C07281=1059.069,212.928,410.818,172.562,33.057,156.142
C07282=1059.063,212.678,410.844,172.560,33.053,156.141
C07283=1059.056,212.430,410.870,172.558,33.049,156.141
C07284=1059.050,212.181,410.896,172.556,33.045,156.140
C07285=1059.045,211.932,410.922,172.554,33.041,156.139
C07286=1059.038,211.684,410.948,172.552,33.037,156.138
C07287=1059.032,211.436,410.973,172.550,33.033,156.138
C07288=1059.026,211.187,411.000,172.548,33.029,156.137
C07289=1059.020,210.939,411.025,172.546,33.026,156.136
C07290=1059.013,210.690,411.051,172.544,33.022,156.135
C07291=1059.007,210.441,411.077,172.542,33.018,156.135
C07292=1059.001,210.192,411.103,172.540,33.014,156.134
C07293=1058.995,209.944,411.129,172.538,33.010,156.133
C07294=1058.988,209.696,411.154,172.536,33.006,156.132
C07295=1058.983,209.447,411.180,172.534,33.002,156.132
C07296=1058.976,209.199,411.206,172.532,32.998,156.131
C07297=1058.970,208.950,411.231,172.530,32.994,156.130
C07298=1058.965,208.717,411.256,172.529,32.990,156.130
C07299=1058.959,208.484,411.280,172.527,32.986,156.129
C07300=1058.954,208.252,411.304,172.525,32.983,156.128
C07301=1058.947,208.020,411.328,172.523,32.979,156.127
C07302=1058.941,207.788,411.352,172.521,32.975,156.127
C07303=1058.936,207.555,411.376,172.520,32.972,156.126
C07304=1058.930,207.323,411.400,172.518,32.968,156.125
C07305=1058.924,207.090,411.424,172.516,32.964,156.125
C07306=1058.899,206.041,411.528,172.330,32.878,156.114
C07307=1058.893,205.792,411.553,172.327,32.874,156.114
C07308=1058.888,205.543,411.577,172.325,32.871,156.113
C07309=1058.881,205.295,411.602,172.323,32.868,156.113
C07310=1058.875,205.045,411.627,172.320,32.865,156.112
C07311=1058.870,204.797,411.652,172.318,32.862,156.112
C07312=1058.864,204.548,411.677,172.316,32.859,156.111
C07313=1058.858,204.300,411.702,172.313,32.856,156.110
C07314=1058.852,204.051,411.726,172.311,32.853,156.110
C07315=1058.846,203.802,411.750,172.309,32.850,156.109
C07316=1058.840,203.554,411.775,172.306,32.846,156.109
C07317=1058.834,203.304,411.800,172.304,32.843,156.108
C07318=1058.829,203.056,411.824,172.302,32.841,156.108
C07319=1058.823,202.807,411.849,172.299,32.838,156.107
C07320=1058.817,202.559,411.874,172.297,32.834,156.107
C07321=1058.811,202.310,411.898,172.295,32.831,156.106
C07322=1058.805,202.062,411.923,172.292,32.828,156.106
C07323=1058.799,201.812,411.947,172.290,32.825,156.105
C07324=1058.793,201.563,411.972,172.288,32.822,156.105
C07325=1058.787,201.315,411.996,172.285,32.819,156.104
C07326=1058.781,201.066,412.020,172.283,32.816,156.104
C07327=1058.775,200.818,412.045,172.281,32.813,156.103
C07328=1058.769,200.569,412.069,172.278,32.810,156.103
C07329=1058.763,200.320,412.093,172.276,32.807,156.102
C07330=1058.757,200.071,412.117,172.274,32.804,156.102
C07331=1058.751,199.822,412.142,172.271,32.801,156.101
C07332=1058.745,199.573,412.166,172.269,32.798,156.100
C07333=1058.739,199.325,412.191,172.267,32.796,156.100
C07334=1058.733,199.077,412.215,172.265,32.792,156.099
C07335=1058.727,198.827,412.239,172.262,32.789,156.099
C07336=1058.721,198.579,412.263,172.260,32.787,156.098
C07337=1058.715,198.330,412.288,172.258,32.783,156.098
C07338=1058.709,198.081,412.311,172.255,32.780,156.097
C07339=1058.703,197.832,412.336,172.253,32.778,156.097
C07340=1058.697,197.584,412.360,172.251,32.775,156.096
C07341=1058.691,197.335,412.384,172.248,32.771,156.096
C07342=1058.685,197.086,412.408,172.247,32.769,156.095
C07343=1058.679,196.837,412.432,172.245,32.766,156.095
C07344=1058.674,196.588,412.457,172.243,32.762,156.094
C07345=1058.668,196.339,412.481,172.240,32.760,156.094
C07346=1058.662,196.091,412.505,172.238,32.757,156.093
C07347=1058.656,195.843,412.529,172.236,32.754,156.093
C07348=1058.650,195.593,412.553,172.234,32.751,156.092
C07349=1058.644,195.345,412.577,172.231,32.748,156.092
C07350=1058.638,195.096,412.602,172.229,32.745,156.091
C07351=1058.632,194.847,412.625,172.227,32.742,156.091
C07352=1058.626,194.598,412.650,172.224,32.739,156.090
C07353=1058.620,194.350,412.674,172.222,32.736,156.090
C07354=1058.615,194.101,412.698,172.220,32.733,156.089
C07355=1058.608,193.852,412.722,172.218,32.730,156.089
C07356=1058.603,193.604,412.746,172.215,32.727,156.088
C07357=1058.597,193.355,412.770,172.213,32.724,156.088
C07358=1058.592,193.106,412.794,172.211,32.722,156.087
C07359=1058.586,192.857,412.817,172.209,32.718,156.087
C07360=1058.579,192.608,412.841,172.207,32.715,156.086
C07361=1058.574,192.360,412.866,172.204,32.713,156.086
C07362=1058.568,192.111,412.889,172.202,32.709,156.085
C07363=1058.562,191.862,412.914,172.200,32.707,156.085
C07364=1058.556,191.613,412.937,172.198,32.704,156.084
C07365=1058.551,191.365,412.961,172.195,32.700,156.084
C07366=1058.544,191.116,412.985,172.193,32.698,156.083
C07367=1058.538,190.832,413.012,172.191,32.695,156.083
C07368=1058.531,190.548,413.040,172.188,32.691,156.082
C07369=1058.525,190.265,413.066,172.186,32.688,156.081
C07370=1058.518,189.981,413.094,172.184,32.684,156.081
C07371=1058.511,189.732,413.118,172.182,32.681,156.080
C07372=1058.507,189.483,413.142,172.180,32.679,156.080
C07373=1058.500,189.235,413.165,172.177,32.675,156.079
C07374=1058.494,188.986,413.189,172.175,32.672,156.079
C07375=1058.489,188.736,413.213,172.173,32.670,156.078
C07376=1058.483,188.488,413.237,172.171,32.667,156.078
C07377=1058.478,188.240,413.261,172.169,32.664,156.077
C07378=1058.471,187.990,413.284,172.166,32.661,156.077
C07379=1058.466,187.741,413.308,172.164,32.658,156.076
C07380=1058.460,187.493,413.332,172.162,32.655,156.076
C07381=1058.454,187.244,413.355,172.160,32.652,156.075
C07382=1058.449,186.996,413.379,172.158,32.649,156.075
C07383=1058.442,186.746,413.403,172.156,32.646,156.074
C07384=1058.437,186.497,413.427,172.153,32.644,156.074
C07385=1058.431,186.249,413.450,172.151,32.640,156.073
C07386=1058.425,186.000,413.473,172.149,32.638,156.073
C07387=1058.420,185.752,413.498,172.147,32.635,156.072
C07388=1058.414,185.502,413.521,172.145,32.631,156.072
C07389=1058.408,185.253,413.545,172.143,32.629,156.071
C07390=1058.403,185.005,413.568,172.140,32.626,156.071
C07391=1058.397,184.756,413.592,172.138,32.623,156.070
C07392=1058.392,184.507,413.615,172.136,32.620,156.070
C07393=1058.385,184.258,413.639,172.134,32.617,156.069
C07394=1058.379,184.009,413.662,172.133,32.614,156.069
C07395=1058.373,183.761,413.686,172.131,32.612,156.068
C07396=1058.367,183.511,413.709,172.128,32.609,156.068
C07397=1058.361,183.262,413.732,172.126,32.606,156.068
C07398=1058.355,183.014,413.756,172.124,32.603,156.067
C07399=1058.349,182.765,413.779,172.122,32.601,156.067
C07400=1058.343,182.516,413.802,172.120,32.598,156.066
C07401=1058.336,182.268,413.825,172.118,32.595,156.066
C07402=1058.331,182.019,413.848,172.115,32.592,156.065
C07403=1058.325,181.770,413.871,172.113,32.590,156.065
C07404=1058.318,181.521,413.895,172.111,32.587,156.064
C07405=1058.313,181.272,413.918,172.109,32.584,156.064
C07406=1058.307,181.023,413.941,172.107,32.581,156.063
C07407=1058.301,180.775,413.965,172.105,32.579,156.063
C07408=1058.294,180.525,413.988,172.102,32.576,156.063
C07409=1058.289,180.276,414.011,172.100,32.573,156.062
C07410=1058.283,180.027,414.034,172.098,32.570,156.062
C07411=1058.276,179.779,414.057,172.096,32.568,156.061
C07412=1058.270,179.531,414.080,172.094,32.565,156.061
C07413=1058.264,179.281,414.103,172.092,32.562,156.060
C07414=1058.258,179.032,414.126,172.090,32.559,156.060
C07415=1058.252,178.784,414.150,172.088,32.557,156.059
C07416=1058.247,178.535,414.173,172.086,32.554,156.059
C07417=1058.241,178.286,414.196,172.084,32.551,156.058
C07418=1058.235,178.037,414.219,172.082,32.548,156.058
C07419=1058.228,177.788,414.241,172.080,32.546,156.057
C07420=1058.222,177.539,414.264,172.078,32.543,156.057
C07421=1058.216,177.291,414.288,172.076,32.540,156.056
C07422=1058.211,177.042,414.311,172.073,32.537,156.056
C07423=1058.205,176.793,414.334,172.071,32.535,156.056
C07424=1058.199,176.544,414.357,172.069,32.532,156.055
C07425=1058.193,176.295,414.380,172.067,32.529,156.055
C07426=1058.186,176.046,414.403,172.065,32.527,156.054
C07427=1058.181,175.797,414.426,172.063,32.524,156.054
C07428=1058.175,175.548,414.448,172.061,32.521,156.053
C07429=1058.169,175.299,414.471,172.059,32.518,156.053
C07430=1058.163,175.050,414.494,172.057,32.516,156.052
C07431=1058.156,174.766,414.521,172.054,32.512,156.052
C07432=1058.149,174.482,414.546,172.052,32.509,156.051
C07433=1058.143,174.198,414.573,172.050,32.506,156.051
C07434=1058.137,173.914,414.599,172.048,32.503,156.050
C07435=1058.131,173.665,414.622,172.046,32.500,156.050
C07436=1058.125,173.416,414.645,172.044,32.498,156.049
C07437=1058.118,173.167,414.667,172.042,32.495,156.049
C07438=1058.112,172.918,414.690,172.040,32.492,156.048
C07439=1058.107,172.669,414.713,172.038,32.489,156.048
C07440=1058.101,172.420,414.736,172.036,32.487,156.047
C07441=1058.095,172.171,414.759,172.034,32.483,156.047
C07442=1058.089,171.923,414.781,172.031,32.481,156.047
C07443=1058.083,171.674,414.804,172.029,32.478,156.046
C07444=1058.077,171.425,414.827,172.027,32.476,156.046
C07445=1058.071,171.176,414.850,172.025,32.472,156.045
C07446=1058.066,170.927,414.873,172.023,32.470,156.045
C07447=1058.059,170.679,414.896,172.021,32.467,156.044
C07448=1058.054,170.429,414.918,172.019,32.465,156.044
C07449=1058.048,170.180,414.941,172.017,32.461,156.043
C07450=1058.042,169.931,414.964,172.015,32.459,156.043
C07451=1058.037,169.682,414.987,172.014,32.456,156.042
C07452=1058.031,169.435,415.009,172.012,32.454,156.042
C07453=1058.025,169.186,415.032,172.010,32.451,156.041
C07454=1058.020,168.936,415.054,172.008,32.448,156.041
C07455=1058.014,168.687,415.077,172.006,32.445,156.041
C07456=1058.007,168.439,415.099,172.004,32.443,156.040
C07457=1058.002,168.190,415.122,172.002,32.440,156.040
C07458=1057.996,167.941,415.145,172.000,32.437,156.039
C07459=1057.991,167.691,415.167,171.998,32.434,156.039
C07460=1057.985,167.442,415.190,171.996,32.432,156.038
C07461=1057.978,167.194,415.213,171.994,32.429,156.038
C07462=1057.973,166.945,415.235,171.992,32.426,156.037
C07463=1057.967,166.695,415.258,171.989,32.423,156.037
C07464=1057.962,166.447,415.280,171.987,32.421,156.036
C07465=1057.956,166.199,415.303,171.985,32.418,156.036
C07466=1057.950,165.949,415.325,171.983,32.415,156.036
C07467=1057.944,165.700,415.348,171.982,32.412,156.035
C07468=1057.938,165.452,415.370,171.980,32.410,156.035
C07469=1057.933,165.202,415.392,171.978,32.407,156.034
C07470=1057.927,164.953,415.415,171.976,32.404,156.034
C07471=1057.921,164.704,415.438,171.974,32.401,156.033
C07472=1057.916,164.456,415.460,171.972,32.399,156.033
C07473=1057.910,164.207,415.483,171.970,32.396,156.032
C07474=1057.904,163.958,415.505,171.968,32.393,156.032
C07475=1057.899,163.709,415.528,171.966,32.391,156.031
C07476=1057.892,163.460,415.550,171.964,32.388,156.031
C07477=1057.887,163.212,415.573,171.962,32.385,156.030
C07478=1057.882,162.962,415.595,171.960,32.382,156.030
C07479=1057.875,162.714,415.617,171.958,32.380,156.030
C07480=1057.870,162.464,415.639,171.956,32.376,156.029
C07481=1057.864,162.215,415.662,171.954,32.374,156.029
C07482=1057.859,161.966,415.684,171.952,32.371,156.028
C07483=1057.853,161.718,415.707,171.952,32.369,156.028
C07484=1057.847,161.468,415.729,171.950,32.366,156.027
C07485=1057.842,161.219,415.752,171.948,32.363,156.027
C07486=1057.835,160.970,415.773,171.946,32.360,156.026
C07487=1057.830,160.722,415.796,171.944,32.358,156.026
C07488=1057.824,160.473,415.818,171.942,32.355,156.025
C07489=1057.818,160.224,415.841,171.940,32.353,156.025
C07490=1057.812,159.975,415.862,171.938,32.350,156.025
C07491=1057.806,159.726,415.885,171.936,32.347,156.024
C07492=1057.800,159.477,415.907,171.934,32.344,156.024
C07493=1057.795,159.228,415.928,171.932,32.342,156.023
C07494=1057.788,158.980,415.950,171.930,32.339,156.023
C07495=1057.782,158.694,415.975,171.927,32.336,156.022
C07496=1057.775,158.410,416.001,171.925,32.333,156.022
C07497=1057.768,158.126,416.027,171.924,32.330,156.021
C07498=1057.762,157.841,416.051,171.922,32.327,156.021
C07499=1057.756,157.592,416.073,171.920,32.325,156.020
C07500=1057.749,157.343,416.095,171.918,32.322,156.020
C07501=1057.744,157.094,416.118,171.916,32.319,156.020
C07502=1057.738,156.845,416.139,171.914,32.317,156.019
C07503=1057.732,156.597,416.161,171.912,32.314,156.019
C07504=1057.726,156.347,416.183,171.910,32.311,156.018
C07505=1057.720,156.098,416.205,171.908,32.309,156.018
C07506=1057.714,155.849,416.227,171.906,32.306,156.017
C07507=1057.709,155.601,416.249,171.904,32.303,156.017
C07508=1057.703,155.351,416.271,171.902,32.301,156.016
C07509=1057.697,155.102,416.293,171.900,32.298,156.016
C07510=1057.691,154.853,416.314,171.898,32.296,156.016
C07511=1057.685,154.605,416.337,171.897,32.293,156.015
C07512=1057.679,154.356,416.358,171.895,32.290,156.015
C07513=1057.673,154.106,416.380,171.893,32.288,156.014
C07514=1057.667,153.857,416.402,171.891,32.285,156.014
C07515=1057.661,153.609,416.423,171.889,32.282,156.013
C07516=1057.656,153.360,416.446,171.887,32.280,156.013
C07517=1057.649,153.111,416.467,171.885,32.277,156.013
C07518=1057.643,152.861,416.489,171.883,32.275,156.012
C07519=1057.638,152.613,416.510,171.882,32.272,156.012
C07520=1057.632,152.364,416.532,171.880,32.270,156.011
C07521=1057.625,152.114,416.554,171.878,32.267,156.011
C07522=1057.620,151.865,416.576,171.876,32.264,156.010
C07523=1057.614,151.616,416.597,171.874,32.262,156.010
C07524=1057.608,151.368,416.620,171.872,32.259,156.010
C07525=1057.602,151.119,416.641,171.871,32.257,156.009
C07526=1057.596,150.870,416.662,171.869,32.254,156.009
C07527=1057.590,150.621,416.684,171.867,32.251,156.008
C07528=1057.585,150.371,416.706,171.865,32.249,156.008
C07529=1057.579,150.123,416.728,171.863,32.246,156.007
C07530=1057.573,149.874,416.749,171.861,32.244,156.007
C07531=1057.567,149.625,416.771,171.859,32.241,156.007
C07532=1057.561,149.376,416.792,171.857,32.238,156.006
C07533=1057.555,149.127,416.814,171.856,32.236,156.006
C07534=1057.549,148.878,416.835,171.854,32.233,156.005
C07535=1057.543,148.629,416.857,171.852,32.231,156.005
C07536=1057.537,148.380,416.878,171.850,32.228,156.004
C07537=1057.531,148.131,416.900,171.848,32.225,156.004
C07538=1057.526,147.882,416.922,171.846,32.223,156.004
C07539=1057.520,147.633,416.943,171.845,32.220,156.003
C07540=1057.514,147.383,416.965,171.843,32.218,156.003
C07541=1057.508,147.135,416.986,171.841,32.215,156.002
C07542=1057.502,146.885,417.007,171.839,32.212,156.002
C07543=1057.495,146.636,417.028,171.837,32.210,156.002
C07544=1057.490,146.388,417.050,171.835,32.207,156.001
C07545=1057.484,146.139,417.071,171.834,32.205,156.001
C07546=1057.478,145.890,417.092,171.832,32.202,156.000
C07547=1057.472,145.641,417.114,171.830,32.199,156.000
C07548=1057.466,145.392,417.136,171.828,32.197,155.999
C07549=1057.460,145.143,417.157,171.826,32.195,155.999
C07550=1057.454,144.893,417.178,171.824,32.192,155.999
C07551=1057.448,144.644,417.200,171.823,32.190,155.998
C07552=1057.443,144.396,417.221,171.821,32.187,155.998
C07553=1057.437,144.146,417.242,171.819,32.184,155.997
C07554=1057.431,143.898,417.264,171.817,32.182,155.997
C07555=1057.424,143.648,417.284,171.816,32.179,155.997
C07556=1057.418,143.399,417.306,171.814,32.177,155.996
C07557=1057.413,143.151,417.327,171.812,32.174,155.996
C07558=1057.407,142.901,417.349,171.810,32.171,155.995
C07559=1057.401,142.616,417.372,171.808,32.169,155.995
C07560=1057.394,142.332,417.397,171.806,32.166,155.994
C07561=1057.386,142.047,417.421,171.803,32.163,155.994
C07562=1057.380,141.763,417.446,171.801,32.160,155.993
C07563=1057.374,141.513,417.467,171.800,32.157,155.993
C07564=1057.368,141.265,417.487,171.799,32.155,155.992
C07565=1057.362,141.015,417.509,171.797,32.152,155.992
C07566=1057.356,140.766,417.530,171.795,32.149,155.992
C07567=1057.351,140.517,417.551,171.793,32.147,155.991
C07568=1057.344,140.268,417.573,171.791,32.144,155.991
C07569=1057.339,140.019,417.593,171.789,32.142,155.990
C07570=1057.333,139.769,417.615,171.787,32.139,155.990
C07571=1057.327,139.521,417.636,171.786,32.137,155.990
C07572=1057.321,139.271,417.657,171.784,32.134,155.989
C07573=1057.315,139.023,417.678,171.782,32.132,155.989
C07574=1057.309,138.773,417.699,171.780,32.129,155.988
C07575=1057.303,138.525,417.719,171.778,32.126,155.988
C07576=1057.297,138.276,417.741,171.777,32.124,155.987
C07577=1057.292,138.027,417.762,171.775,32.121,155.987
C07578=1057.285,137.777,417.783,171.773,32.119,155.987
C07579=1057.279,137.529,417.803,171.772,32.117,155.986
C07580=1057.273,137.279,417.825,171.770,32.114,155.986
C07581=1057.268,137.030,417.845,171.768,32.111,155.985
C07582=1057.261,136.781,417.867,171.766,32.109,155.985
C07583=1057.256,136.532,417.887,171.764,32.106,155.985
C07584=1057.250,136.283,417.909,171.762,32.104,155.984
C07585=1057.244,136.034,417.929,171.760,32.102,155.984
C07586=1057.238,135.785,417.950,171.759,32.099,155.983
C07587=1057.232,135.536,417.971,171.757,32.096,155.983
C07588=1057.225,135.287,417.992,171.756,32.094,155.983
C07589=1057.220,135.038,418.012,171.754,32.091,155.982
C07590=1057.214,134.789,418.034,171.752,32.089,155.982
C07591=1057.208,134.540,418.054,171.750,32.086,155.981
C07592=1057.202,134.291,418.076,171.749,32.084,155.981
C07593=1057.196,134.042,418.096,171.747,32.081,155.981
C07594=1057.190,133.792,418.117,171.745,32.079,155.980
C07595=1057.184,133.543,418.138,171.743,32.076,155.980
C07596=1057.178,133.295,418.158,171.741,32.074,155.979
C07597=1057.172,133.045,418.179,171.739,32.071,155.979
C07598=1057.167,132.796,418.200,171.738,32.068,155.978
C07599=1057.160,132.547,418.220,171.737,32.066,155.978
C07600=1057.155,132.298,418.242,171.735,32.063,155.978
C07601=1057.149,132.050,418.262,171.733,32.061,155.977
C07602=1057.143,131.800,418.282,171.731,32.059,155.977
C07603=1057.137,131.551,418.304,171.729,32.056,155.976
C07604=1057.131,131.302,418.324,171.728,32.053,155.976
C07605=1057.125,131.053,418.344,171.726,32.051,155.976
C07606=1057.119,130.804,418.366,171.724,32.049,155.975
C07607=1057.113,130.555,418.386,171.722,32.046,155.975
C07608=1057.106,130.305,418.406,171.720,32.044,155.974
C07609=1057.101,130.056,418.426,171.718,32.041,155.974
C07610=1057.094,129.807,418.448,171.717,32.039,155.974
C07611=1057.089,129.558,418.468,171.716,32.036,155.973
C07612=1057.083,129.309,418.488,171.714,32.034,155.973
C07613=1057.076,129.060,418.508,171.712,32.031,155.972
C07614=1057.071,128.811,418.530,171.710,32.029,155.972
C07615=1057.064,128.562,418.550,171.708,32.026,155.972
C07616=1057.058,128.313,418.570,171.707,32.024,155.971
C07617=1057.053,128.064,418.590,171.705,32.021,155.971
C07618=1057.046,127.814,418.611,171.703,32.019,155.971
C07619=1057.040,127.566,418.631,171.701,32.017,155.970
C07620=1057.034,127.316,418.652,171.699,32.014,155.970
C07621=1057.028,127.068,418.672,171.698,32.012,155.969
C07622=1057.022,126.819,418.692,171.697,32.010,155.969
C07623=1057.015,126.533,418.716,171.695,32.006,155.968
C07624=1057.009,126.249,418.739,171.693,32.004,155.968
C07625=1057.002,125.963,418.763,171.690,32.001,155.968
C07626=1056.994,125.679,418.786,171.688,31.998,155.967
C07627=1056.989,125.429,418.806,171.687,31.996,155.967
C07628=1056.983,125.180,418.826,171.685,31.993,155.966
C07629=1056.977,124.931,418.846,171.683,31.991,155.966
C07630=1056.971,124.682,418.867,171.681,31.988,155.965
C07631=1056.965,124.433,418.887,171.679,31.986,155.965
C07632=1056.959,124.184,418.907,171.679,31.983,155.965
C07633=1056.952,123.935,418.928,171.677,31.981,155.964
C07634=1056.947,123.685,418.948,171.675,31.978,155.964
C07635=1056.941,123.437,418.968,171.673,31.975,155.963
C07636=1056.934,123.187,418.988,171.671,31.973,155.963
C07637=1056.929,122.938,419.009,171.670,31.971,155.963
C07638=1056.923,122.689,419.029,171.668,31.968,155.962
C07639=1056.916,122.440,419.049,171.666,31.966,155.962
C07640=1056.911,122.190,419.070,171.664,31.963,155.961
C07641=1056.905,121.942,419.090,171.662,31.961,155.961
C07642=1056.899,121.693,419.110,171.661,31.958,155.961
C07643=1056.893,121.443,419.130,171.660,31.956,155.960
C07644=1056.887,121.194,419.151,171.658,31.953,155.960
C07645=1056.881,120.945,419.171,171.656,31.951,155.959
C07646=1056.875,120.697,419.191,171.655,31.949,155.959
C07647=1056.869,120.447,419.211,171.653,31.946,155.959
C07648=1056.863,120.198,419.231,171.651,31.943,155.958
C07649=1056.857,119.949,419.251,171.649,31.941,155.958
C07650=1056.851,119.700,419.271,171.647,31.938,155.957
C07651=1056.846,119.450,419.292,171.646,31.936,155.957
C07652=1056.840,119.202,419.312,171.644,31.934,155.957
C07653=1056.834,118.952,419.331,171.643,31.931,155.956
C07654=1056.828,118.703,419.351,171.641,31.928,155.956
C07655=1056.822,118.454,419.372,171.640,31.926,155.955
C07656=1056.816,118.205,419.392,171.638,31.923,155.955
C07657=1056.810,117.956,419.412,171.636,31.921,155.955
C07658=1056.804,117.707,419.432,171.634,31.918,155.954
C07659=1056.799,117.458,419.453,171.633,31.916,155.954
C07660=1056.793,117.209,419.472,171.631,31.913,155.953
C07661=1056.787,116.959,419.492,171.629,31.911,155.953
C07662=1056.781,116.710,419.512,171.627,31.908,155.953
C07663=1056.775,116.461,419.532,171.626,31.906,155.952
C07664=1056.769,116.212,419.553,171.625,31.904,155.952
C07665=1056.764,115.963,419.572,171.623,31.901,155.951
C07666=1056.758,115.714,419.592,171.621,31.898,155.951
C07667=1056.751,115.465,419.612,171.620,31.896,155.951
C07668=1056.746,115.215,419.633,171.618,31.893,155.950
C07669=1056.740,114.966,419.652,171.616,31.891,155.950
C07670=1056.734,114.717,419.672,171.614,31.888,155.949
C07671=1056.728,114.468,419.692,171.613,31.886,155.949
C07672=1056.723,114.219,419.713,171.611,31.883,155.949
C07673=1056.717,113.970,419.732,171.610,31.881,155.948
C07674=1056.711,113.720,419.752,171.608,31.878,155.948
C07675=1056.705,113.472,419.772,171.606,31.876,155.947
C07676=1056.699,113.222,419.791,171.605,31.873,155.947
C07677=1056.693,112.973,419.811,171.603,31.871,155.947
C07678=1056.687,112.724,419.831,171.601,31.869,155.946
C07679=1056.681,112.475,419.851,171.599,31.866,155.946
C07680=1056.675,112.226,419.871,171.598,31.864,155.945
C07681=1056.669,111.977,419.891,171.596,31.861,155.945
C07682=1056.663,111.727,419.910,171.594,31.859,155.945
C07683=1056.657,111.478,419.930,171.593,31.856,155.944
C07684=1056.651,111.229,419.949,171.592,31.854,155.944
C07685=1056.645,110.980,419.969,171.590,31.851,155.943
C07686=1056.638,110.730,419.988,171.588,31.849,155.943
C07687=1056.632,110.446,420.012,171.586,31.846,155.943
C07688=1056.625,110.161,420.033,171.584,31.843,155.942
C07689=1056.618,109.876,420.055,171.582,31.841,155.942
C07690=1056.610,109.591,420.079,171.580,31.838,155.941
C07691=1056.605,109.341,420.098,171.578,31.835,155.941
C07692=1056.599,109.092,420.118,171.577,31.833,155.941
C07693=1056.593,108.843,420.137,171.576,31.831,155.940
C07694=1056.587,108.594,420.157,171.574,31.828,155.940
C07695=1056.581,108.345,420.176,171.572,31.825,155.939
C07696=1056.575,108.096,420.196,171.571,31.823,155.939
C07697=1056.569,107.847,420.215,171.569,31.821,155.939
C07698=1056.562,107.597,420.235,171.567,31.818,155.938
C07699=1056.557,107.348,420.254,171.565,31.816,155.938
C07700=1056.551,107.098,420.274,171.564,31.814,155.937
C07701=1056.544,106.850,420.293,171.562,31.811,155.937
C07702=1056.539,106.600,420.312,171.561,31.809,155.937
C07703=1056.533,106.352,420.332,171.560,31.806,155.936
C07704=1056.527,106.102,420.351,171.558,31.804,155.936
C07705=1056.521,105.853,420.371,171.556,31.801,155.935
C07706=1056.514,105.604,420.390,171.554,31.799,155.935
C07707=1056.509,105.355,420.409,171.553,31.797,155.935
C07708=1056.503,105.106,420.429,171.551,31.794,155.934
C07709=1056.497,104.857,420.448,171.549,31.792,155.934
C07710=1056.491,104.607,420.468,171.547,31.789,155.934
C07711=1056.485,104.359,420.487,171.546,31.787,155.933
C07712=1056.478,104.109,420.507,171.545,31.784,155.933
C07713=1056.473,103.859,420.526,171.543,31.782,155.932
C07714=1056.467,103.610,420.546,171.541,31.779,155.932
C07715=1056.461,103.361,420.565,171.540,31.777,155.932
C07716=1056.455,103.112,420.584,171.538,31.775,155.931
C07717=1056.449,102.863,420.604,171.536,31.772,155.931
C07718=1056.443,102.613,420.623,171.535,31.770,155.930
C07719=1056.437,102.364,420.642,171.533,31.767,155.930
C07720=1056.431,102.115,420.662,171.531,31.765,155.930
C07721=1056.425,101.866,420.681,171.530,31.762,155.929
C07722=1056.419,101.617,420.700,171.529,31.760,155.929
C07723=1056.413,101.367,420.719,171.527,31.757,155.928
C07724=1056.407,101.118,420.739,171.525,31.755,155.928
C07725=1056.401,100.869,420.758,171.524,31.752,155.928
C07726=1056.395,100.620,420.777,171.522,31.750,155.927
C07727=1056.390,100.370,420.796,171.520,31.748,155.927
C07728=1056.383,100.122,420.816,171.518,31.745,155.927
C07729=1056.377,99.873,420.835,171.517,31.743,155.926
C07730=1056.371,99.623,420.854,171.516,31.741,155.926
C07731=1056.365,99.374,420.873,171.514,31.738,155.925
C07732=1056.359,99.125,420.892,171.513,31.736,155.925
C07733=1056.353,98.875,420.911,171.511,31.733,155.925
C07734=1056.347,98.626,420.929,171.509,31.731,155.924
C07735=1056.341,98.377,420.949,171.507,31.729,155.924
C07736=1056.334,98.128,420.968,171.506,31.726,155.924
C07737=1056.328,97.879,420.987,171.504,31.723,155.923
C07738=1056.323,97.629,421.007,171.502,31.721,155.923
C07739=1056.316,97.380,421.025,171.501,31.719,155.922
C07740=1056.311,97.131,421.044,171.500,31.716,155.922
C07741=1056.305,96.883,421.063,171.498,31.714,155.922
C07742=1056.299,96.633,421.082,171.496,31.711,155.921
C07743=1056.293,96.384,421.101,171.495,31.710,155.921
C07744=1056.287,96.135,421.120,171.493,31.707,155.921
C07745=1056.280,95.886,421.139,171.491,31.704,155.920
C07746=1056.275,95.637,421.158,171.489,31.702,155.920
C07747=1056.268,95.387,421.177,171.488,31.700,155.919
C07748=1056.262,95.138,421.196,171.487,31.697,155.919
C07749=1056.256,94.889,421.215,171.485,31.695,155.919
C07750=1056.250,94.639,421.234,171.484,31.692,155.918
C07751=1056.244,94.354,421.255,171.482,31.690,155.918
C07752=1056.236,94.069,421.277,171.480,31.687,155.917
C07753=1056.229,93.784,421.299,171.478,31.684,155.917
C07754=1056.223,93.499,421.321,171.476,31.681,155.916
C07755=1056.216,93.250,421.339,171.474,31.679,155.916
C07756=1056.211,93.001,421.358,171.473,31.676,155.916
C07757=1056.205,92.752,421.376,171.472,31.674,155.915
C07758=1056.199,92.502,421.396,171.470,31.671,155.915
C07759=1056.193,92.253,421.414,171.468,31.669,155.915
C07760=1056.187,92.004,421.433,171.467,31.667,155.914
C07761=1056.181,91.755,421.452,171.465,31.664,155.914
C07762=1056.175,91.505,421.471,171.463,31.662,155.913
C07763=1056.169,91.257,421.490,171.462,31.659,155.913
C07764=1056.164,91.007,421.509,171.460,31.657,155.913
C07765=1056.157,90.758,421.527,171.459,31.655,155.912
C07766=1056.151,90.509,421.547,171.457,31.652,155.912
C07767=1056.145,90.260,421.565,171.456,31.650,155.911
C07768=1056.139,90.010,421.583,171.454,31.647,155.911
C07769=1056.132,89.761,421.602,171.452,31.645,155.911
C07770=1056.127,89.511,421.621,171.451,31.643,155.910
C07771=1056.120,89.262,421.640,171.449,31.640,155.910
C07772=1056.114,89.014,421.658,171.447,31.638,155.910
C07773=1056.108,88.764,421.676,171.445,31.635,155.909
C07774=1056.103,88.515,421.695,171.445,31.633,155.909
C07775=1056.096,88.265,421.714,171.443,31.631,155.909
C07776=1056.090,88.016,421.733,171.441,31.628,155.908
C07777=1056.083,87.767,421.751,171.440,31.626,155.908
C07778=1056.078,87.517,421.770,171.438,31.624,155.907
C07779=1056.072,87.269,421.788,171.436,31.622,155.907
C07780=1056.066,87.020,421.807,171.435,31.619,155.907
C07781=1056.059,86.770,421.825,171.433,31.616,155.906
C07782=1056.053,86.521,421.843,171.432,31.614,155.906
C07783=1056.048,86.271,421.863,171.430,31.612,155.906
C07784=1056.041,86.022,421.881,171.429,31.610,155.905
C07785=1056.036,85.773,421.899,171.427,31.607,155.905
C07786=1056.029,85.524,421.917,171.425,31.604,155.904
C07787=1056.023,85.275,421.937,171.424,31.602,155.904
C07788=1056.017,85.025,421.955,171.422,31.600,155.904
C07789=1056.011,84.776,421.973,171.420,31.598,155.903
C07790=1056.005,84.527,421.992,171.419,31.595,155.903
C07791=1055.999,84.278,422.010,171.418,31.593,155.903
C07792=1055.993,84.028,422.029,171.416,31.590,155.902
C07793=1055.987,83.779,422.047,171.415,31.588,155.902
C07794=1055.981,83.529,422.065,171.413,31.586,155.902
C07795=1055.975,83.281,422.084,171.411,31.583,155.901
C07796=1055.969,83.032,422.102,171.409,31.581,155.901
C07797=1055.962,82.782,422.120,171.408,31.579,155.900
C07798=1055.957,82.533,422.139,171.406,31.576,155.900
C07799=1055.951,82.284,422.158,171.405,31.574,155.900
C07800=1055.945,82.034,422.176,171.404,31.571,155.899
C07801=1055.938,81.785,422.194,171.402,31.569,155.899
C07802=1055.932,81.536,422.212,171.400,31.567,155.899
C07803=1055.927,81.287,422.231,171.399,31.564,155.898
C07804=1055.921,81.037,422.249,171.397,31.561,155.898
C07805=1055.915,80.788,422.268,171.395,31.559,155.897
C07806=1055.909,80.539,422.286,171.394,31.557,155.897
C07807=1055.903,80.290,422.304,171.393,31.555,155.897
C07808=1055.896,80.041,422.323,171.391,31.552,155.896
C07809=1055.891,79.791,422.341,171.390,31.550,155.896
C07810=1055.885,79.542,422.359,171.388,31.547,155.896
C07811=1055.879,79.292,422.377,171.386,31.545,155.895
C07812=1055.872,79.043,422.396,171.384,31.542,155.895
C07813=1055.867,78.794,422.413,171.383,31.540,155.894
C07814=1055.861,78.545,422.432,171.381,31.537,155.894
C07815=1055.853,78.260,422.453,171.380,31.535,155.894
C07816=1055.847,77.975,422.474,171.378,31.532,155.893
C07817=1055.840,77.690,422.494,171.376,31.529,155.893
C07818=1055.833,77.404,422.515,171.374,31.527,155.892
C07819=1055.827,77.155,422.533,171.373,31.524,155.892
C07820=1055.821,76.906,422.551,171.371,31.522,155.892
C07821=1055.815,76.656,422.569,171.369,31.520,155.891
C07822=1055.808,76.407,422.588,171.368,31.518,155.891
C07823=1055.803,76.158,422.605,171.367,31.515,155.890
C07824=1055.797,75.909,422.623,171.365,31.513,155.890
C07825=1055.790,75.659,422.642,171.364,31.510,155.890
C07826=1055.785,75.410,422.660,171.362,31.508,155.889
C07827=1055.779,75.161,422.677,171.360,31.506,155.889
C07828=1055.772,74.911,422.696,171.359,31.503,155.889
C07829=1055.766,74.663,422.713,171.357,31.501,155.888
C07830=1055.760,74.413,422.731,171.355,31.498,155.888
C07831=1055.753,74.164,422.750,171.354,31.496,155.888
C07832=1055.748,73.915,422.767,171.353,31.494,155.887
C07833=1055.742,73.665,422.785,171.351,31.492,155.887
C07834=1055.735,73.416,422.804,171.349,31.489,155.886
C07835=1055.730,73.167,422.821,171.348,31.487,155.886
C07836=1055.724,72.917,422.839,171.346,31.484,155.886
C07837=1055.718,72.667,422.857,171.344,31.482,155.885
C07838=1055.712,72.419,422.876,171.343,31.480,155.885
C07839=1055.706,72.169,422.893,171.342,31.477,155.885
C07840=1055.699,71.920,422.911,171.340,31.475,155.884
C07841=1055.693,71.671,422.928,171.339,31.472,155.884
C07842=1055.687,71.422,422.947,171.337,31.470,155.884
C07843=1055.681,71.173,422.965,171.335,31.468,155.883
C07844=1055.675,70.923,422.983,171.334,31.466,155.883
C07845=1055.669,70.673,423.000,171.332,31.463,155.882
C07846=1055.663,70.425,423.019,171.331,31.461,155.882
C07847=1055.656,70.175,423.036,171.330,31.458,155.882
C07848=1055.651,69.926,423.054,171.328,31.456,155.881
C07849=1055.645,69.677,423.072,171.326,31.454,155.881
C07850=1055.639,69.427,423.089,171.324,31.451,155.881
C07851=1055.633,69.178,423.107,171.323,31.449,155.880
C07852=1055.626,68.928,423.124,171.321,31.446,155.880
C07853=1055.620,68.680,423.143,171.319,31.444,155.880
C07854=1055.614,68.430,423.161,171.319,31.442,155.879
C07855=1055.608,68.180,423.179,171.317,31.440,155.879
C07856=1055.602,67.932,423.196,171.315,31.437,155.878
C07857=1055.596,67.682,423.213,171.314,31.435,155.878
C07858=1055.590,67.433,423.231,171.312,31.432,155.878
C07859=1055.583,67.184,423.248,171.310,31.430,155.877
C07860=1055.578,66.934,423.266,171.309,31.428,155.877
C07861=1055.572,66.685,423.284,171.307,31.426,155.877
C07862=1055.566,66.435,423.302,171.306,31.423,155.876
C07863=1055.559,66.187,423.319,171.305,31.421,155.876
C07864=1055.553,65.937,423.337,171.303,31.418,155.876
C07865=1055.547,65.688,423.355,171.301,31.416,155.875
C07866=1055.541,65.439,423.372,171.299,31.414,155.875
C07867=1055.535,65.190,423.390,171.298,31.412,155.875
C07868=1055.529,64.940,423.408,171.296,31.409,155.874
C07869=1055.523,64.691,423.425,171.295,31.407,155.874
C07870=1055.517,64.441,423.443,171.294,31.404,155.873
C07871=1055.510,64.192,423.461,171.292,31.402,155.873
C07872=1055.504,63.943,423.478,171.290,31.400,155.873
C07873=1055.498,63.693,423.496,171.289,31.398,155.872
C07874=1055.492,63.444,423.512,171.287,31.395,155.872
C07875=1055.485,63.194,423.529,171.285,31.393,155.872
C07876=1055.480,62.945,423.547,171.284,31.391,155.871
C07877=1055.473,62.696,423.564,171.283,31.389,155.871
C07878=1055.467,62.446,423.582,171.281,31.386,155.871
C07879=1055.459,62.162,423.602,171.279,31.383,155.870
C07880=1055.452,61.876,423.622,171.277,31.381,155.870
C07881=1055.446,61.591,423.641,171.275,31.379,155.870
C07882=1055.438,61.306,423.661,171.273,31.376,155.869
C07883=1055.432,61.057,423.679,171.272,31.373,155.869
C07884=1055.426,60.807,423.695,171.271,31.371,155.868
C07885=1055.420,60.558,423.712,171.269,31.369,155.868
C07886=1055.414,60.308,423.730,171.268,31.367,155.868
C07887=1055.407,60.059,423.748,171.266,31.365,155.867
C07888=1055.401,59.810,423.765,171.264,31.362,155.867
C07889=1055.394,59.560,423.783,171.263,31.360,155.867
C07890=1055.388,59.311,423.799,171.261,31.358,155.866
C07891=1055.382,59.061,423.817,171.259,31.355,155.866
C07892=1055.376,58.813,423.834,171.258,31.353,155.866
C07893=1055.370,58.563,423.852,171.257,31.351,155.865
C07894=1055.364,58.314,423.869,171.255,31.348,155.865
C07895=1055.358,58.065,423.885,171.253,31.346,155.865
C07896=1055.352,57.815,423.903,171.252,31.344,155.864
C07897=1055.345,57.566,423.920,171.250,31.342,155.864
C07898=1055.339,57.316,423.938,171.248,31.339,155.864
C07899=1055.333,57.067,423.954,171.248,31.337,155.863
C07900=1055.326,56.818,423.971,171.246,31.334,155.863
C07901=1055.321,56.569,423.989,171.244,31.332,155.863
C07902=1055.314,56.319,424.006,171.243,31.330,155.862
C07903=1055.309,56.070,424.023,171.241,31.328,155.862
C07904=1055.302,55.820,424.040,171.239,31.326,155.862
C07905=1055.296,55.571,424.057,171.237,31.323,155.861
C07906=1055.290,55.322,424.074,171.236,31.321,155.861
C07907=1055.284,55.072,424.092,171.235,31.319,155.861
C07908=1055.277,54.824,424.109,171.233,31.316,155.860
C07909=1055.271,54.573,424.126,171.232,31.314,155.860
C07910=1055.265,54.325,424.143,171.230,31.312,155.859
C07911=1055.259,54.075,424.161,171.228,31.309,155.859
C07912=1055.253,53.825,424.177,171.227,31.307,155.859
C07913=1055.247,53.577,424.194,171.225,31.305,155.858
C07914=1055.241,53.327,424.212,171.224,31.303,155.858
C07915=1055.235,53.078,424.228,171.223,31.300,155.858
C07916=1055.229,52.829,424.245,171.221,31.298,155.857
C07917=1055.222,52.579,424.263,171.219,31.295,155.857
C07918=1055.216,52.330,424.279,171.217,31.293,155.857
C07919=1055.210,52.080,424.297,171.216,31.291,155.856
C07920=1055.204,51.831,424.314,171.214,31.289,155.856
C07921=1055.198,51.582,424.330,171.213,31.286,155.856
C07922=1055.192,51.332,424.347,171.212,31.284,155.855
C07923=1055.186,51.083,424.365,171.210,31.282,155.855
C07924=1055.180,50.834,424.382,171.208,31.279,155.855
C07925=1055.173,50.584,424.398,171.207,31.277,155.854
C07926=1055.168,50.335,424.416,171.205,31.275,155.854
C07927=1055.162,50.086,424.432,171.203,31.272,155.854
C07928=1055.155,49.836,424.449,171.203,31.270,155.853
C07929=1055.150,49.587,424.466,171.201,31.268,155.853
C07930=1055.143,49.338,424.483,171.199,31.265,155.852
C07931=1055.137,49.088,424.500,171.198,31.263,155.852
C07932=1055.131,48.839,424.517,171.196,31.261,155.852
C07933=1055.125,48.589,424.534,171.194,31.258,155.851
C07934=1055.119,48.341,424.551,171.192,31.256,155.851
C07935=1055.113,48.090,424.568,171.192,31.254,155.851
C07936=1055.107,47.842,424.585,171.190,31.252,155.850
C07937=1055.101,47.592,424.601,171.188,31.249,155.850
C07938=1055.094,47.343,424.618,171.187,31.247,155.850
C07939=1055.089,47.093,424.635,171.185,31.244,155.849
C07940=1055.083,46.844,424.652,171.183,31.242,155.849
C07941=1055.077,46.595,424.669,171.182,31.240,155.849
C07942=1055.071,46.345,424.686,171.181,31.238,155.848
C07943=1055.064,46.060,424.705,171.179,31.235,155.848
C07944=1055.058,45.775,424.724,171.177,31.232,155.847
C07945=1055.050,45.488,424.743,171.175,31.229,155.847
C07946=1055.044,45.203,424.763,171.173,31.227,155.847
C07947=1055.038,44.954,424.779,171.172,31.225,155.846
C07948=1055.031,44.704,424.796,171.171,31.222,155.846
C07949=1055.026,44.455,424.813,171.169,31.220,155.846
C07950=1055.020,44.205,424.829,171.167,31.217,155.845
C07951=1055.014,43.957,424.846,171.166,31.215,155.845
C07952=1055.007,43.707,424.863,171.164,31.213,155.845
C07953=1055.002,43.457,424.880,171.162,31.211,155.844
C07954=1054.996,43.208,424.897,171.161,31.208,155.844
C07955=1054.990,42.959,424.913,171.160,31.206,155.844
C07956=1054.983,42.709,424.930,171.158,31.204,155.843
C07957=1054.977,42.460,424.947,171.157,31.201,155.843
C07958=1054.971,42.211,424.963,171.155,31.199,155.843
C07959=1054.965,41.961,424.979,171.153,31.197,155.842
C07960=1054.958,41.711,424.996,171.151,31.194,155.842
C07961=1054.952,41.463,425.013,171.150,31.192,155.842
C07962=1054.946,41.213,425.029,171.149,31.190,155.841
C07963=1054.940,40.964,425.045,171.147,31.188,155.841
C07964=1054.934,40.715,425.061,171.146,31.186,155.840
C07965=1054.928,40.464,425.078,171.144,31.184,155.840
C07966=1054.921,40.216,425.095,171.142,31.181,155.840
C07967=1054.916,39.966,425.111,171.141,31.179,155.839
C07968=1054.910,39.717,425.128,171.139,31.177,155.839
C07969=1054.904,39.468,425.144,171.138,31.174,155.839
C07970=1054.897,39.218,425.160,171.136,31.172,155.839
C07971=1054.891,38.969,425.177,171.135,31.169,155.838
C07972=1054.885,38.720,425.194,171.133,31.167,155.838
C07973=1054.879,38.470,425.210,171.131,31.165,155.838
C07974=1054.874,38.221,425.227,171.130,31.163,155.837
C07975=1054.868,37.971,425.243,171.128,31.161,155.837
C07976=1054.861,37.721,425.260,171.127,31.158,155.837
C07977=1054.855,37.472,425.275,171.125,31.156,155.836
C07978=1054.849,37.223,425.292,171.124,31.154,155.836
C07979=1054.842,36.974,425.308,171.122,31.152,155.835
C07980=1054.836,36.725,425.325,171.120,31.150,155.835
C07981=1054.830,36.475,425.341,171.119,31.147,155.835
C07982=1054.824,36.225,425.358,171.117,31.145,155.834
C07983=1054.817,35.976,425.373,171.116,31.143,155.834
C07984=1054.811,35.727,425.390,171.114,31.141,155.834
C07985=1054.805,35.478,425.406,171.113,31.138,155.833
C07986=1054.799,35.228,425.422,171.111,31.136,155.833
C07987=1054.793,34.978,425.439,171.109,31.134,155.833
C07988=1054.787,34.729,425.455,171.108,31.132,155.833
C07989=1054.780,34.480,425.471,171.107,31.129,155.832
C07990=1054.774,34.230,425.487,171.105,31.127,155.832
C07991=1054.768,33.981,425.503,171.103,31.125,155.832
C07992=1054.762,33.732,425.519,171.102,31.123,155.831
C07993=1054.756,33.482,425.536,171.100,31.120,155.831
C07994=1054.749,33.233,425.552,171.098,31.118,155.831
C07995=1054.743,32.983,425.568,171.097,31.116,155.830
C07996=1054.737,32.734,425.584,171.096,31.114,155.830
C07997=1054.731,32.485,425.600,171.094,31.111,155.830
C07998=1054.725,32.235,425.617,171.092,31.109,155.829
C07999=1054.719,31.986,425.632,171.091,31.107,155.829
C08000=1054.713,31.736,425.648,171.089,31.105,155.829
C08001=1054.707,31.487,425.664,171.087,31.103,155.828
C08002=1054.700,31.237,425.681,171.085,31.100,155.828
C08003=1054.694,30.988,425.697,171.085,31.098,155.828
C08004=1054.688,30.738,425.713,171.083,31.096,155.827
C08005=1054.682,30.489,425.729,171.081,31.094,155.827
C08006=1054.676,30.240,425.745,171.080,31.092,155.827
C08007=1054.669,29.954,425.763,171.078,31.089,155.826
C08008=1054.662,29.669,425.782,171.076,31.086,155.826
C08009=1054.655,29.383,425.800,171.075,31.084,155.826
C08010=1054.648,29.097,425.819,171.073,31.081,155.825
C08011=1054.641,28.848,425.834,171.071,31.079,155.825
C08012=1054.635,28.599,425.851,171.069,31.077,155.825
C08013=1054.629,28.349,425.867,171.068,31.075,155.824
C08014=1054.623,28.100,425.882,171.066,31.073,155.824
C08015=1054.617,27.850,425.898,171.064,31.070,155.824
C08016=1054.611,27.601,425.914,171.063,31.068,155.823
C08017=1054.604,27.352,425.930,171.062,31.066,155.823
C08018=1054.599,27.102,425.946,171.060,31.064,155.823
C08019=1054.593,26.853,425.962,171.058,31.062,155.822
C08020=1054.586,26.603,425.977,171.056,31.059,155.822
C08021=1054.580,26.354,425.994,171.055,31.057,155.822
C08022=1054.574,26.105,426.009,171.054,31.055,155.821
C08023=1054.568,25.855,426.025,171.052,31.053,155.821
C08024=1054.562,25.606,426.041,171.050,31.051,155.821
C08025=1054.555,25.357,426.057,171.049,31.049,155.821
C08026=1054.549,25.106,426.073,171.047,31.046,155.820
C08027=1054.542,24.857,426.088,171.045,31.044,155.820
C08028=1054.536,24.608,426.105,171.043,31.042,155.820
C08029=1054.530,24.358,426.120,171.043,31.040,155.819
C08030=1054.524,24.109,426.136,171.041,31.038,155.819
C08031=1054.517,23.860,426.151,171.039,31.035,155.819
C08032=1054.512,23.610,426.167,171.037,31.033,155.818
C08033=1054.506,23.360,426.183,171.036,31.031,155.818
C08034=1054.499,23.111,426.199,171.034,31.029,155.818
C08035=1054.493,22.861,426.214,171.033,31.027,155.817
C08036=1054.487,22.612,426.230,171.032,31.025,155.817
C08037=1054.481,22.363,426.246,171.030,31.022,155.817
C08038=1054.474,22.113,426.261,171.028,31.020,155.816
C08039=1054.469,21.865,426.277,171.026,31.018,155.816
C08040=1054.463,21.615,426.292,171.025,31.016,155.816
C08041=1054.457,21.366,426.308,171.023,31.014,155.815
C08042=1054.450,21.117,426.324,171.022,31.011,155.815
C08043=1054.444,20.867,426.340,171.020,31.009,155.815
C08044=1054.438,20.618,426.355,171.019,31.007,155.815
C08045=1054.432,20.368,426.371,171.017,31.005,155.814
C08046=1054.426,20.118,426.387,171.015,31.002,155.814
C08047=1054.420,19.869,426.402,171.013,31.000,155.814
C08048=1054.413,19.620,426.418,171.013,30.998,155.813
C08049=1054.407,19.370,426.433,171.011,30.996,155.813
C08050=1054.401,19.121,426.449,171.009,30.994,155.813
C08051=1054.395,18.871,426.464,171.007,30.992,155.812
C08052=1054.388,18.622,426.480,171.006,30.990,155.812
C08053=1054.382,18.372,426.495,171.004,30.987,155.812
C08054=1054.376,18.123,426.511,171.002,30.985,155.811
C08055=1054.370,17.873,426.526,171.001,30.983,155.811
C08056=1054.364,17.624,426.543,170.999,30.981,155.811
C08057=1054.357,17.374,426.557,170.998,30.979,155.811
C08058=1054.352,17.125,426.572,170.996,30.977,155.810
C08059=1054.346,16.876,426.588,170.994,30.975,155.810
C08060=1054.339,16.626,426.603,170.992,30.973,155.810
C08061=1054.333,16.377,426.620,170.991,30.971,155.809
C08062=1054.327,16.127,426.634,170.990,30.968,155.809
C08063=1054.320,15.878,426.650,170.988,30.966,155.809
C08064=1054.315,15.628,426.666,170.986,30.964,155.808
C08065=1054.308,15.378,426.681,170.985,30.962,155.808
C08066=1054.301,15.129,426.696,170.983,30.960,155.808
C08067=1054.296,14.880,426.711,170.981,30.958,155.808
C08068=1054.290,14.630,426.726,170.980,30.955,155.807
C08069=1054.284,14.381,426.743,170.979,30.953,155.807
C08070=1054.278,14.131,426.758,170.977,30.951,155.807
C08071=1054.271,13.847,426.775,170.975,30.949,155.806
C08072=1054.263,13.563,426.792,170.973,30.946,155.806
C08073=1054.256,13.279,426.810,170.971,30.944,155.806
C08074=1054.249,12.994,426.827,170.970,30.942,155.805
C08075=1054.243,12.745,426.842,170.968,30.939,155.805
C08076=1054.236,12.496,426.858,170.966,30.937,155.805
C08077=1054.229,12.246,426.873,170.964,30.935,155.804
C08078=1054.224,11.996,426.888,170.963,30.933,155.804
C08079=1054.217,11.746,426.903,170.961,30.931,155.804
C08080=1054.211,11.498,426.918,170.960,30.929,155.804
C08081=1054.205,11.248,426.933,170.958,30.927,155.803
C08082=1054.199,10.999,426.948,170.956,30.925,155.803
C08083=1054.192,10.749,426.963,170.955,30.923,155.803
C08084=1054.186,10.499,426.978,170.953,30.921,155.802
C08085=1054.179,10.250,426.994,170.951,30.919,155.802
C08086=1054.173,10.000,427.009,170.949,30.916,155.802
C08087=1054.168,9.751,427.024,170.948,30.915,155.802
C08088=1054.161,9.502,427.039,170.947,30.913,155.801
C08089=1054.155,9.252,427.054,170.945,30.911,155.801
C08090=1054.148,9.003,427.069,170.943,30.909,155.801
C08091=1054.142,8.753,427.084,170.941,30.907,155.801
C08092=1054.135,8.504,427.099,170.940,30.905,155.800
C08093=1054.130,8.255,427.114,170.939,30.902,155.800
C08094=1054.124,8.005,427.129,170.937,30.900,155.800
C08095=1054.118,7.755,427.144,170.935,30.898,155.799
C08096=1054.111,7.505,427.159,170.933,30.896,155.799
C08097=1054.105,7.256,427.174,170.932,30.894,155.799
C08098=1054.099,7.007,427.190,170.930,30.892,155.799
C08099=1054.092,6.758,427.205,170.928,30.890,155.798
C08100=1054.086,6.508,427.219,170.927,30.888,155.798
C08101=1054.080,6.258,427.234,170.925,30.886,155.798
C08102=1054.074,6.010,427.249,170.924,30.884,155.797
C08103=1054.067,5.760,427.264,170.922,30.882,155.797
C08104=1054.062,5.510,427.279,170.920,30.879,155.797
C08105=1054.055,5.260,427.294,170.918,30.877,155.797
C08106=1054.050,5.011,427.309,170.917,30.875,155.796
C08107=1054.043,4.762,427.324,170.916,30.873,155.796
C08108=1054.037,4.512,427.339,170.914,30.871,155.796
C08109=1054.031,4.262,427.354,170.912,30.869,155.795
C08110=1054.025,4.013,427.368,170.910,30.867,155.795
C08111=1054.018,3.764,427.383,170.908,30.865,155.795
C08112=1054.012,3.514,427.398,170.908,30.863,155.794
C08113=1054.006,3.264,427.413,170.906,30.861,155.794
C08114=1054.000,3.015,427.428,170.904,30.858,155.794
C08115=1053.993,2.766,427.443,170.902,30.856,155.794
C08116=1053.987,2.516,427.458,170.900,30.855,155.793
C08117=1053.982,2.267,427.473,170.899,30.853,155.793
C08118=1053.976,2.017,427.488,170.897,30.851,155.793
C08119=1053.969,1.768,427.503,170.896,30.849,155.793
C08120=1053.963,1.519,427.517,170.894,30.846,155.792
C08121=1053.957,1.269,427.532,170.892,30.844,155.792
C08122=1053.951,1.019,427.547,170.891,30.842,155.792
C08123=1053.945,0.770,427.562,170.889,30.840,155.791
C08124=1053.939,0.521,427.577,170.887,30.838,155.791
C08125=1053.932,0.270,427.591,170.886,30.836,155.791
C08126=1053.927,0.021,427.606,170.884,30.834,155.791
C08127=1053.920,-0.228,427.621,170.883,30.832,155.790
C08128=1053.914,-0.478,427.635,170.881,30.830,155.790
C08129=1053.908,-0.727,427.650,170.879,30.827,155.790
C08130=1053.902,-0.977,427.665,170.877,30.825,155.789
C08131=1053.895,-1.226,427.680,170.876,30.823,155.789
C08132=1053.890,-1.475,427.695,170.874,30.821,155.789
C08133=1053.883,-1.725,427.709,170.873,30.819,155.789
C08134=1053.878,-1.974,427.723,170.871,30.817,155.788
C08135=1053.870,-2.257,427.740,170.869,30.815,155.788
C08136=1053.864,-2.539,427.757,170.867,30.813,155.788
C08137=1053.857,-2.821,427.774,170.866,30.810,155.787
C08138=1053.850,-3.104,427.790,170.864,30.808,155.787
C08139=1053.844,-3.354,427.805,170.862,30.806,155.787
C08140=1053.838,-3.603,427.819,170.860,30.804,155.787
C08141=1053.832,-3.853,427.834,170.858,30.802,155.786
C08142=1053.825,-4.102,427.848,170.856,30.800,155.786
C08143=1053.819,-4.351,427.862,170.855,30.798,155.786
C08144=1053.813,-4.601,427.877,170.854,30.796,155.785
C08145=1053.806,-4.850,427.892,170.852,30.794,155.785
C08146=1053.800,-5.100,427.906,170.850,30.792,155.785
C08147=1053.794,-5.350,427.921,170.848,30.790,155.785
C08148=1053.788,-5.599,427.935,170.846,30.788,155.784
C08149=1053.781,-5.849,427.949,170.845,30.786,155.784
C08150=1053.775,-6.098,427.964,170.844,30.784,155.784
C08151=1053.769,-6.347,427.978,170.842,30.782,155.784
C08152=1053.763,-6.597,427.993,170.840,30.780,155.783
C08153=1053.756,-6.847,428.007,170.838,30.778,155.783
C08154=1053.750,-7.096,428.022,170.836,30.776,155.783
C08155=1053.744,-7.346,428.036,170.835,30.774,155.783
C08156=1053.737,-7.595,428.050,170.833,30.772,155.782
C08157=1053.731,-7.845,428.064,170.832,30.770,155.782
C08158=1053.726,-8.094,428.079,170.830,30.769,155.782
C08159=1053.719,-8.344,428.093,170.828,30.766,155.782
C08160=1053.712,-8.594,428.107,170.826,30.764,155.781
C08161=1053.707,-8.843,428.122,170.824,30.762,155.781
C08162=1053.700,-9.093,428.136,170.823,30.761,155.781
C08163=1053.694,-9.341,428.150,170.821,30.759,155.781
C08164=1053.688,-9.592,428.164,170.820,30.757,155.780
C08165=1053.682,-9.841,428.179,170.818,30.754,155.780
C08166=1053.675,-10.090,428.193,170.816,30.753,155.780
C08167=1053.670,-10.340,428.207,170.814,30.751,155.780
C08168=1053.663,-10.589,428.222,170.813,30.749,155.779
C08169=1053.658,-10.839,428.236,170.811,30.746,155.779
C08170=1053.651,-11.088,428.250,170.809,30.745,155.779
C08171=1053.645,-11.338,428.264,170.808,30.743,155.779
C08172=1053.639,-11.587,428.279,170.806,30.741,155.778
C08173=1053.632,-11.837,428.292,170.804,30.739,155.778
C08174=1053.626,-12.086,428.307,170.803,30.737,155.778
C08175=1053.621,-12.336,428.321,170.801,30.735,155.778
C08176=1053.613,-12.585,428.335,170.799,30.733,155.777
C08177=1053.608,-12.835,428.349,170.797,30.731,155.777
C08178=1053.602,-13.085,428.363,170.796,30.729,155.777
C08179=1053.595,-13.334,428.377,170.794,30.727,155.777
C08180=1053.589,-13.584,428.392,170.793,30.725,155.776
C08181=1053.584,-13.833,428.406,170.791,30.724,155.776
C08182=1053.577,-14.083,428.420,170.789,30.721,155.776
C08183=1053.571,-14.332,428.434,170.787,30.719,155.776
C08184=1053.564,-14.582,428.448,170.785,30.717,155.775
C08185=1053.559,-14.831,428.462,170.784,30.716,155.775
C08186=1053.552,-15.081,428.477,170.782,30.714,155.775
C08187=1053.546,-15.330,428.490,170.781,30.711,155.775
C08188=1053.540,-15.581,428.504,170.779,30.710,155.774
C08189=1053.533,-15.829,428.518,170.777,30.708,155.774
C08190=1053.528,-16.079,428.532,170.775,30.706,155.774
C08191=1053.521,-16.329,428.546,170.773,30.704,155.774
C08192=1053.515,-16.577,428.560,170.771,30.702,155.773
C08193=1053.509,-16.828,428.574,170.770,30.700,155.773
C08194=1053.502,-17.077,428.587,170.769,30.698,155.773
C08195=1053.496,-17.327,428.602,170.767,30.697,155.773
C08196=1053.490,-17.576,428.616,170.765,30.695,155.772
C08197=1053.484,-17.826,428.630,170.763,30.693,155.772
C08198=1053.477,-18.075,428.643,170.761,30.691,155.772
C08199=1053.472,-18.301,428.657,170.760,30.689,155.772
C08200=1053.466,-18.526,428.669,170.759,30.687,155.772
C08201=1053.460,-18.752,428.681,170.757,30.686,155.771
C08202=1053.455,-18.977,428.693,170.755,30.684,155.771
C08203=1053.449,-19.204,428.706,170.753,30.682,155.771
C08204=1053.443,-19.429,428.719,170.752,30.681,155.771
C08205=1053.438,-19.655,428.731,170.750,30.679,155.771
C08206=1053.432,-19.881,428.743,170.749,30.677,155.770
C08207=1053.426,-20.130,428.758,170.747,30.676,155.770
C08208=1053.420,-20.379,428.771,170.745,30.674,155.770
C08209=1053.413,-20.629,428.785,170.744,30.672,155.770
C08210=1053.408,-20.878,428.799,170.742,30.670,155.769
C08211=1053.401,-21.128,428.812,170.740,30.668,155.769
C08212=1053.395,-21.378,428.826,170.738,30.666,155.769
C08213=1053.389,-21.627,428.840,170.737,30.665,155.769
C08214=1053.382,-21.877,428.854,170.735,30.663,155.768
C08215=1053.377,-22.126,428.868,170.733,30.661,155.768
C08216=1053.370,-22.375,428.881,170.731,30.659,155.768
C08217=1053.364,-22.626,428.895,170.729,30.657,155.768
C08218=1053.358,-22.875,428.908,170.727,30.655,155.768
C08219=1053.352,-23.124,428.922,170.727,30.653,155.767
C08220=1053.346,-23.375,428.936,170.725,30.652,155.767
C08221=1053.339,-23.623,428.950,170.723,30.650,155.767
C08222=1053.333,-23.872,428.963,170.721,30.648,155.767
C08223=1053.327,-24.123,428.977,170.719,30.646,155.766
C08224=1053.321,-24.372,428.991,170.717,30.644,155.766
C08225=1053.315,-24.622,429.005,170.716,30.642,155.766
C08226=1053.308,-24.872,429.018,170.714,30.641,155.766
C08227=1053.302,-25.121,429.032,170.712,30.638,155.766
C08228=1053.297,-25.370,429.045,170.710,30.637,155.765
C08229=1053.290,-25.620,429.059,170.708,30.635,155.765
C08230=1053.284,-25.870,429.072,170.707,30.633,155.765
C08231=1053.278,-26.119,429.086,170.705,30.631,155.765
C08232=1053.272,-26.368,429.099,170.704,30.630,155.764
C08233=1053.265,-26.618,429.113,170.702,30.628,155.764
C08234=1053.260,-26.868,429.127,170.700,30.625,155.764
C08235=1053.253,-27.117,429.140,170.698,30.624,155.764
C08236=1053.247,-27.367,429.154,170.696,30.622,155.764
C08237=1053.240,-27.616,429.167,170.694,30.620,155.763
C08238=1053.234,-27.866,429.180,170.693,30.619,155.763
C08239=1053.227,-28.116,429.194,170.691,30.617,155.763
C08240=1053.222,-28.365,429.208,170.689,30.615,155.763
C08241=1053.216,-28.615,429.221,170.687,30.613,155.763
C08242=1053.210,-28.864,429.234,170.685,30.612,155.762
C08243=1053.203,-29.114,429.247,170.683,30.610,155.762
C08244=1053.197,-29.364,429.261,170.682,30.608,155.762
C08245=1053.191,-29.613,429.274,170.681,30.606,155.762
C08246=1053.184,-29.862,429.287,170.679,30.605,155.761
C08247=1053.178,-30.112,429.301,170.677,30.603,155.761
C08248=1053.171,-30.361,429.314,170.675,30.601,155.761
C08249=1053.166,-30.611,429.328,170.673,30.599,155.761
C08250=1053.159,-30.861,429.342,170.671,30.598,155.761
C08251=1053.153,-31.111,429.354,170.670,30.596,155.760
C08252=1053.147,-31.360,429.367,170.668,30.594,155.760
C08253=1053.141,-31.609,429.381,170.666,30.593,155.760
C08254=1053.135,-31.859,429.394,170.664,30.590,155.760
C08255=1053.126,-32.188,429.412,170.661,30.588,155.760
C08256=1053.118,-32.517,429.428,170.660,30.586,155.759
C08257=1053.110,-32.845,429.446,170.657,30.584,155.759
C08258=1053.101,-33.173,429.463,170.655,30.581,155.759
C08259=1053.096,-33.423,429.477,170.653,30.580,155.759
C08260=1053.089,-33.673,429.491,170.651,30.578,155.758
C08261=1053.083,-33.923,429.503,170.649,30.576,155.758
C08262=1053.077,-34.172,429.517,170.648,30.575,155.758
C08263=1053.070,-34.452,429.532,170.646,30.573,155.758
C08264=1053.063,-34.732,429.546,170.644,30.571,155.758
C08265=1053.056,-35.012,429.561,170.641,30.569,155.757
C08266=1053.049,-35.292,429.575,170.639,30.566,155.757
C08267=1053.043,-35.542,429.589,170.637,30.565,155.757
C08268=1053.037,-35.791,429.602,170.636,30.563,155.757
C08269=1053.030,-36.041,429.615,170.634,30.562,155.757
C08270=1053.024,-36.290,429.628,170.632,30.560,155.756
C08271=1053.018,-36.539,429.641,170.630,30.558,155.756
C08272=1053.012,-36.789,429.654,170.628,30.557,155.756
C08273=1053.006,-37.038,429.667,170.626,30.554,155.756
C08274=1053.001,-37.289,429.680,170.625,30.553,155.756
C08275=1052.994,-37.539,429.694,170.624,30.552,155.755
C08276=1052.988,-37.788,429.707,170.622,30.549,155.755
C08277=1052.982,-38.038,429.720,170.620,30.548,155.755
C08278=1052.976,-38.287,429.733,170.618,30.546,155.755
C08279=1052.969,-38.536,429.746,170.616,30.545,155.755
C08280=1052.963,-38.786,429.759,170.614,30.543,155.754
C08281=1052.956,-39.035,429.772,170.613,30.541,155.754
C08282=1052.951,-39.285,429.784,170.611,30.539,155.754
C08283=1052.944,-39.535,429.798,170.609,30.538,155.754
C08284=1052.938,-39.785,429.810,170.607,30.536,155.754
C08285=1052.932,-40.034,429.824,170.605,30.535,155.754
C08286=1052.926,-40.284,429.836,170.603,30.533,155.753
C08287=1052.919,-40.533,429.849,170.601,30.532,155.753
C08288=1052.913,-40.783,429.861,170.600,30.530,155.753
C08289=1052.907,-41.032,429.875,170.598,30.528,155.753
C08290=1052.901,-41.282,429.887,170.596,30.526,155.753
C08291=1052.895,-41.531,429.901,170.594,30.525,155.752
C08292=1052.888,-41.782,429.914,170.592,30.523,155.752
C08293=1052.881,-42.031,429.926,170.590,30.522,155.752
C08294=1052.875,-42.281,429.939,170.589,30.520,155.752
C08295=1052.869,-42.530,429.952,170.587,30.519,155.752
C08296=1052.863,-42.780,429.965,170.585,30.516,155.752
C08297=1052.857,-43.029,429.978,170.583,30.515,155.751
C08298=1052.850,-43.279,429.990,170.581,30.513,155.751
C08299=1052.844,-43.528,430.002,170.579,30.512,155.751
C08300=1052.838,-43.778,430.016,170.577,30.510,155.751
C08301=1052.832,-44.028,430.028,170.576,30.509,155.751
C08302=1052.826,-44.277,430.041,170.574,30.507,155.751
C08303=1052.819,-44.526,430.053,170.572,30.506,155.750
C08304=1052.813,-44.776,430.066,170.570,30.504,155.750
C08305=1052.807,-45.026,430.079,170.568,30.503,155.750
C08306=1052.801,-45.275,430.092,170.566,30.501,155.750
C08307=1052.794,-45.524,430.104,170.565,30.499,155.750
C08308=1052.788,-45.774,430.117,170.563,30.497,155.749
C08309=1052.782,-46.024,430.130,170.561,30.496,155.749
C08310=1052.776,-46.273,430.143,170.559,30.494,155.749
C08311=1052.770,-46.523,430.155,170.557,30.493,155.749
C08312=1052.764,-46.773,430.167,170.555,30.491,155.749
C08313=1052.757,-47.022,430.181,170.553,30.489,155.749
C08314=1052.752,-47.272,430.193,170.552,30.488,155.749
C08315=1052.746,-47.522,430.206,170.550,30.486,155.748
C08316=1052.739,-47.772,430.218,170.548,30.485,155.748
C08317=1052.733,-48.021,430.231,170.546,30.483,155.748
C08318=1052.727,-48.271,430.243,170.544,30.482,155.748
C08319=1052.721,-48.521,430.256,170.542,30.480,155.748
C08320=1052.714,-48.769,430.269,170.541,30.479,155.748
C08321=1052.708,-49.019,430.281,170.539,30.477,155.747
C08322=1052.702,-49.269,430.294,170.537,30.475,155.747
C08323=1052.696,-49.519,430.306,170.535,30.474,155.747
C08324=1052.690,-49.769,430.318,170.533,30.472,155.747
C08325=1052.683,-50.018,430.332,170.531,30.471,155.747
C08326=1052.678,-50.268,430.344,170.529,30.469,155.747
C08327=1052.671,-50.548,430.357,170.527,30.468,155.746
C08328=1052.664,-50.828,430.371,170.525,30.466,155.746
C08329=1052.656,-51.109,430.385,170.523,30.464,155.746
C08330=1052.649,-51.389,430.400,170.521,30.462,155.746
C08331=1052.643,-51.638,430.412,170.519,30.461,155.746
C08332=1052.637,-51.888,430.424,170.516,30.460,155.746
C08333=1052.630,-52.138,430.436,170.515,30.458,155.746
C08334=1052.624,-52.388,430.449,170.513,30.456,155.745
C08335=1052.618,-52.637,430.461,170.511,30.456,155.745
C08336=1052.611,-52.887,430.473,170.509,30.454,155.745
C08337=1052.605,-53.137,430.485,170.507,30.452,155.745
C08338=1052.598,-53.386,430.497,170.505,30.451,155.745
C08339=1052.592,-53.636,430.510,170.503,30.449,155.745
C08340=1052.586,-53.886,430.522,170.502,30.448,155.745
C08341=1052.580,-54.135,430.535,170.500,30.447,155.744
C08342=1052.573,-54.385,430.547,170.498,30.445,155.744
C08343=1052.566,-54.634,430.559,170.496,30.444,155.744
C08344=1052.560,-54.884,430.571,170.494,30.443,155.744
C08345=1052.554,-55.133,430.583,170.492,30.441,155.744
C08346=1052.548,-55.383,430.595,170.490,30.440,155.744
C08347=1052.542,-55.632,430.607,170.489,30.438,155.744
C08348=1052.535,-55.882,430.619,170.487,30.437,155.744
C08349=1052.529,-56.132,430.632,170.485,30.436,155.743
C08350=1052.523,-56.381,430.644,170.483,30.434,155.743
C08351=1052.516,-56.631,430.656,170.481,30.432,155.743
C08352=1052.510,-56.881,430.668,170.479,30.431,155.743
C08353=1052.504,-57.131,430.680,170.476,30.430,155.743
C08354=1052.498,-57.380,430.692,170.475,30.428,155.743
C08355=1052.492,-57.630,430.704,170.473,30.427,155.743
C08356=1052.485,-57.879,430.716,170.471,30.426,155.743
C08357=1052.479,-58.129,430.728,170.469,30.424,155.742
C08358=1052.473,-58.379,430.740,170.467,30.423,155.742
C08359=1052.466,-58.628,430.752,170.465,30.421,155.742
C08360=1052.460,-58.878,430.765,170.463,30.420,155.742
C08361=1052.454,-59.127,430.776,170.462,30.418,155.742
C08362=1052.448,-59.377,430.789,170.460,30.417,155.742
C08363=1052.441,-59.627,430.801,170.458,30.416,155.742
C08364=1052.435,-59.877,430.812,170.456,30.414,155.742
C08365=1052.429,-60.127,430.825,170.454,30.413,155.741
C08366=1052.423,-60.376,430.836,170.452,30.412,155.741
C08367=1052.416,-60.625,430.848,170.450,30.410,155.741
C08368=1052.411,-60.875,430.861,170.448,30.409,155.741
C08369=1052.404,-61.125,430.873,170.447,30.408,155.741
C08370=1052.397,-61.374,430.885,170.444,30.406,155.741
C08371=1052.392,-61.624,430.896,170.442,30.405,155.741
C08372=1052.386,-61.873,430.908,170.440,30.404,155.741
C08373=1052.379,-62.123,430.920,170.438,30.402,155.740
C08374=1052.373,-62.373,430.933,170.436,30.400,155.740
C08375=1052.367,-62.622,430.944,170.434,30.400,155.740
C08376=1052.361,-62.872,430.955,170.433,30.398,155.740
C08377=1052.355,-63.122,430.968,170.431,30.396,155.740
C08378=1052.348,-63.371,430.980,170.429,30.395,155.740
C08379=1052.342,-63.620,430.992,170.427,30.394,155.740
C08380=1052.336,-63.871,431.003,170.425,30.392,155.740
C08381=1052.330,-64.120,431.015,170.423,30.391,155.740
C08382=1052.323,-64.370,431.027,170.421,30.390,155.739
C08383=1052.317,-64.619,431.038,170.420,30.388,155.739
C08384=1052.312,-64.869,431.051,170.417,30.387,155.739
C08385=1052.305,-65.119,431.063,170.415,30.386,155.739
C08386=1052.299,-65.368,431.074,170.413,30.385,155.739
C08387=1052.293,-65.618,431.086,170.411,30.383,155.739
C08388=1052.287,-65.868,431.098,170.409,30.381,155.739
C08389=1052.281,-66.117,431.110,170.407,30.381,155.739
C08390=1052.275,-66.367,431.122,170.406,30.379,155.738
C08391=1052.267,-66.649,431.135,170.404,30.377,155.738
C08392=1052.261,-66.930,431.148,170.401,30.376,155.738
C08393=1052.254,-67.212,431.162,170.399,30.375,155.738
C08394=1052.246,-67.493,431.174,170.397,30.373,155.738
C08395=1052.241,-67.744,431.186,170.395,30.372,155.738
C08396=1052.235,-67.993,431.198,170.393,30.370,155.738
C08397=1052.228,-68.243,431.209,170.391,30.369,155.738
C08398=1052.223,-68.493,431.222,170.389,30.368,155.738
C08399=1052.217,-68.742,431.233,170.387,30.366,155.737
C08400=1052.210,-68.992,431.245,170.385,30.365,155.737
C08401=1052.204,-69.241,431.256,170.383,30.364,155.737
C08402=1052.199,-69.491,431.268,170.381,30.362,155.737
C08403=1052.192,-69.741,431.280,170.379,30.361,155.737
C08404=1052.186,-69.990,431.291,170.378,30.360,155.737
C08405=1052.180,-70.240,431.303,170.376,30.359,155.737
C08406=1052.174,-70.490,431.315,170.374,30.357,155.737
C08407=1052.168,-70.739,431.326,170.372,30.356,155.737
C08408=1052.161,-70.989,431.338,170.369,30.355,155.737
C08409=1052.155,-71.238,431.349,170.367,30.354,155.737
C08410=1052.150,-71.488,431.362,170.365,30.352,155.736
C08411=1052.144,-71.738,431.372,170.364,30.351,155.736
C08412=1052.137,-71.987,431.384,170.362,30.350,155.736
C08413=1052.131,-72.237,431.396,170.360,30.349,155.736
C08414=1052.125,-72.487,431.407,170.358,30.347,155.736
C08415=1052.119,-72.737,431.419,170.356,30.346,155.736
C08416=1052.113,-72.986,431.430,170.354,30.344,155.736
C08417=1052.107,-73.236,431.442,170.352,30.344,155.736
C08418=1052.101,-73.485,431.453,170.350,30.342,155.736
C08419=1052.095,-73.735,431.465,170.348,30.341,155.736
C08420=1052.089,-73.985,431.476,170.346,30.339,155.735
C08421=1052.083,-74.235,431.487,170.344,30.338,155.735
C08422=1052.077,-74.484,431.499,170.342,30.337,155.735
C08423=1052.071,-74.734,431.510,170.340,30.336,155.735
C08424=1052.064,-74.984,431.522,170.338,30.335,155.735
C08425=1052.058,-75.233,431.533,170.336,30.333,155.735
C08426=1052.052,-75.483,431.544,170.335,30.332,155.735
C08427=1052.046,-75.732,431.556,170.333,30.331,155.735
C08428=1052.040,-75.982,431.567,170.330,30.330,155.735
C08429=1052.034,-76.232,431.578,170.328,30.329,155.735
C08430=1052.027,-76.481,431.590,170.326,30.328,155.735
C08431=1052.021,-76.731,431.601,170.324,30.327,155.735
C08432=1052.015,-76.981,431.612,170.322,30.325,155.734
C08433=1052.009,-77.231,431.623,170.320,30.324,155.734
C08434=1052.002,-77.480,431.634,170.319,30.323,155.734
C08435=1051.996,-77.730,431.646,170.317,30.322,155.734
C08436=1051.990,-77.980,431.657,170.314,30.321,155.734
C08437=1051.983,-78.229,431.669,170.312,30.320,155.734
C08438=1051.978,-78.479,431.679,170.310,30.319,155.734
C08439=1051.971,-78.729,431.691,170.308,30.317,155.734
C08440=1051.965,-78.978,431.702,170.306,30.316,155.734
C08441=1051.960,-79.228,431.712,170.304,30.315,155.734
C08442=1051.953,-79.477,431.724,170.303,30.314,155.734
C08443=1051.947,-79.727,431.735,170.301,30.313,155.734
C08444=1051.941,-79.977,431.746,170.298,30.312,155.734
C08445=1051.935,-80.226,431.757,170.296,30.311,155.734
C08446=1051.928,-80.476,431.768,170.294,30.310,155.734
C08447=1051.922,-80.726,431.780,170.292,30.309,155.733
C08448=1051.916,-80.975,431.791,170.290,30.308,155.733
C08449=1051.909,-81.226,431.802,170.288,30.307,155.733
C08450=1051.903,-81.475,431.812,170.287,30.306,155.733
C08451=1051.897,-81.725,431.824,170.284,30.305,155.733
C08452=1051.891,-81.974,431.834,170.282,30.304,155.733
C08453=1051.884,-82.224,431.845,170.280,30.303,155.733
C08454=1051.878,-82.474,431.856,170.278,30.302,155.733
C08455=1051.871,-82.758,431.869,170.276,30.300,155.733
C08456=1051.864,-83.042,431.881,170.273,30.299,155.733
C08457=1051.857,-83.326,431.894,170.271,30.298,155.733
C08458=1051.850,-83.609,431.906,170.269,30.297,155.733
C08459=1051.843,-83.859,431.917,170.267,30.296,155.733
C08460=1051.838,-84.109,431.928,170.265,30.295,155.733
C08461=1051.831,-84.358,431.938,170.263,30.294,155.733
C08462=1051.825,-84.608,431.949,170.261,30.293,155.733
C08463=1051.819,-84.858,431.961,170.259,30.292,155.733
C08464=1051.812,-85.107,431.971,170.256,30.291,155.733
C08465=1051.806,-85.358,431.982,170.254,30.290,155.733
C08466=1051.800,-85.607,431.993,170.253,30.289,155.733
C08467=1051.794,-85.856,432.004,170.251,30.288,155.733
C08468=1051.787,-86.106,432.014,170.249,30.287,155.733
C08469=1051.781,-86.356,432.025,170.247,30.286,155.733
C08470=1051.775,-86.606,432.037,170.245,30.285,155.733
C08471=1051.769,-86.855,432.047,170.242,30.284,155.733
C08472=1051.763,-87.105,432.058,170.240,30.283,155.732
C08473=1051.757,-87.355,432.069,170.238,30.282,155.732
C08474=1051.750,-87.604,432.079,170.236,30.281,155.732
C08475=1051.744,-87.854,432.090,170.235,30.280,155.732
C08476=1051.738,-88.104,432.101,170.233,30.279,155.732
C08477=1051.731,-88.353,432.112,170.230,30.278,155.732
C08478=1051.726,-88.602,432.123,170.228,30.277,155.732
C08479=1051.719,-88.853,432.134,170.226,30.276,155.732
C08480=1051.713,-89.102,432.144,170.224,30.275,155.732
C08481=1051.708,-89.352,432.154,170.222,30.274,155.732
C08482=1051.701,-89.602,432.165,170.220,30.274,155.732
C08483=1051.695,-89.851,432.176,170.218,30.272,155.732
C08484=1051.689,-90.101,432.187,170.216,30.271,155.732
C08485=1051.683,-90.351,432.198,170.214,30.270,155.732
C08486=1051.676,-90.600,432.208,170.212,30.270,155.732
C08487=1051.670,-90.850,432.219,170.210,30.269,155.732
C08488=1051.664,-91.100,432.229,170.208,30.268,155.732
C08489=1051.658,-91.350,432.240,170.206,30.267,155.732
C08490=1051.652,-91.599,432.251,170.203,30.266,155.732
C08491=1051.645,-91.849,432.261,170.201,30.265,155.732
C08492=1051.639,-92.098,432.272,170.200,30.264,155.732
C08493=1051.634,-92.349,432.282,170.198,30.263,155.732
C08494=1051.627,-92.598,432.293,170.196,30.262,155.732
C08495=1051.621,-92.848,432.304,170.194,30.261,155.732
C08496=1051.615,-93.097,432.314,170.191,30.261,155.732
C08497=1051.609,-93.347,432.325,170.189,30.260,155.732
C08498=1051.603,-93.597,432.335,170.187,30.259,155.732
C08499=1051.596,-93.847,432.346,170.185,30.258,155.732
C08500=1051.591,-94.096,432.357,170.183,30.257,155.732
C08501=1051.584,-94.346,432.366,170.182,30.256,155.732
C08502=1051.579,-94.595,432.377,170.179,30.255,155.732
C08503=1051.573,-94.845,432.388,170.177,30.255,155.732
C08504=1051.566,-95.095,432.399,170.175,30.254,155.732
C08505=1051.560,-95.345,432.409,170.173,30.253,155.732
C08506=1051.554,-95.594,432.419,170.171,30.252,155.732
C08507=1051.548,-95.844,432.430,170.169,30.251,155.731
C08508=1051.543,-96.094,432.440,170.166,30.250,155.732
C08509=1051.536,-96.344,432.451,170.164,30.249,155.732
C08510=1051.530,-96.593,432.462,170.163,30.248,155.731
C08511=1051.524,-96.843,432.471,170.161,30.247,155.731
C08512=1051.518,-97.092,432.482,170.159,30.246,155.731
C08513=1051.513,-97.342,432.492,170.157,30.246,155.731
C08514=1051.506,-97.592,432.503,170.154,30.245,155.731
C08515=1051.499,-97.841,432.513,170.152,30.244,155.731
C08516=1051.494,-98.092,432.523,170.150,30.244,155.731
C08517=1051.487,-98.341,432.534,170.148,30.243,155.731
C08518=1051.480,-98.591,432.544,170.146,30.242,155.731
C08519=1051.474,-98.878,432.556,170.144,30.241,155.732
C08520=1051.467,-99.164,432.567,170.142,30.240,155.731
C08521=1051.460,-99.450,432.579,170.139,30.239,155.731
C08522=1051.453,-99.736,432.591,170.137,30.239,155.732
C08523=1051.446,-99.985,432.601,170.135,30.238,155.731
C08524=1051.441,-100.236,432.611,170.132,30.237,155.731
C08525=1051.434,-100.485,432.622,170.130,30.236,155.732
C08526=1051.428,-100.734,432.631,170.128,30.235,155.732
C08527=1051.422,-100.984,432.642,170.126,30.235,155.732
C08528=1051.416,-101.234,432.652,170.124,30.234,155.732
C08529=1051.409,-101.484,432.662,170.122,30.233,155.732
C08530=1051.403,-101.734,432.673,170.120,30.233,155.732
C08531=1051.397,-101.983,432.683,170.118,30.232,155.732
C08532=1051.391,-102.233,432.692,170.116,30.231,155.732
C08533=1051.385,-102.482,432.703,170.114,30.230,155.732
C08534=1051.379,-102.732,432.713,170.111,30.230,155.732
C08535=1051.372,-102.981,432.723,170.109,30.229,155.732
C08536=1051.366,-103.231,432.733,170.107,30.228,155.732
C08537=1051.360,-103.482,432.743,170.105,30.227,155.732
C08538=1051.354,-103.731,432.753,170.103,30.227,155.732
C08539=1051.348,-103.981,432.763,170.102,30.226,155.732
C08540=1051.342,-104.230,432.774,170.099,30.226,155.732
C08541=1051.336,-104.480,432.784,170.097,30.225,155.732
C08542=1051.329,-104.730,432.793,170.095,30.224,155.732
C08543=1051.324,-104.979,432.804,170.093,30.223,155.732
C08544=1051.318,-105.229,432.814,170.091,30.223,155.732
C08545=1051.311,-105.479,432.823,170.088,30.222,155.732
C08546=1051.305,-105.728,432.833,170.086,30.222,155.732
C08547=1051.300,-105.978,432.844,170.084,30.221,155.732
C08548=1051.293,-106.228,432.853,170.082,30.220,155.732
C08549=1051.286,-106.478,432.864,170.081,30.219,155.732
C08550=1051.280,-106.728,432.873,170.078,30.219,155.732
C08551=1051.275,-106.978,432.883,170.076,30.218,155.732
C08552=1051.268,-107.228,432.893,170.074,30.217,155.732
C08553=1051.262,-107.477,432.903,170.072,30.217,155.732
C08554=1051.256,-107.727,432.913,170.070,30.216,155.732
C08555=1051.250,-107.976,432.922,170.067,30.216,155.732
C08556=1051.243,-108.226,432.932,170.065,30.215,155.732
C08557=1051.238,-108.476,432.943,170.063,30.214,155.732
C08558=1051.232,-108.725,432.952,170.061,30.214,155.732
C08559=1051.225,-108.975,432.962,170.059,30.214,155.732
C08560=1051.219,-109.225,432.972,170.057,30.212,155.732
C08561=1051.213,-109.474,432.982,170.055,30.212,155.732
C08562=1051.207,-109.724,432.991,170.053,30.212,155.732
C08563=1051.200,-109.974,433.001,170.051,30.211,155.733
C08564=1051.194,-110.224,433.011,170.049,30.210,155.733
C08565=1051.188,-110.473,433.020,170.046,30.210,155.733
C08566=1051.183,-110.724,433.030,170.044,30.210,155.733
C08567=1051.176,-110.973,433.041,170.042,30.209,155.733
C08568=1051.170,-111.223,433.050,170.040,30.208,155.733
C08569=1051.164,-111.472,433.060,170.037,30.208,155.733
C08570=1051.158,-111.722,433.069,170.035,30.207,155.733
C08571=1051.151,-111.972,433.079,170.033,30.206,155.733
C08572=1051.145,-112.222,433.088,170.032,30.206,155.733
C08573=1051.139,-112.472,433.098,170.030,30.206,155.733
C08574=1051.133,-112.721,433.108,170.027,30.205,155.733
C08575=1051.126,-112.970,433.118,170.025,30.204,155.733
C08576=1051.120,-113.220,433.127,170.023,30.204,155.733
C08577=1051.114,-113.470,433.137,170.021,30.204,155.733
C08578=1051.109,-113.720,433.147,170.019,30.203,155.733
C08579=1051.103,-113.970,433.157,170.016,30.202,155.733
C08580=1051.096,-114.220,433.166,170.014,30.202,155.733
C08581=1051.090,-114.470,433.176,170.012,30.201,155.733
C08582=1051.084,-114.719,433.185,170.010,30.201,155.733
C08583=1051.077,-115.004,433.196,170.007,30.201,155.734
C08584=1051.070,-115.289,433.207,170.006,30.200,155.734
C08585=1051.062,-115.574,433.218,170.003,30.200,155.734
C08586=1051.056,-115.859,433.229,170.001,30.199,155.734
C08587=1051.050,-116.108,433.238,169.998,30.198,155.734
C08588=1051.044,-116.358,433.248,169.996,30.198,155.734
C08589=1051.038,-116.608,433.258,169.994,30.198,155.734
C08590=1051.031,-116.857,433.267,169.992,30.197,155.734
C08591=1051.025,-117.107,433.275,169.990,30.197,155.734
C08592=1051.019,-117.357,433.285,169.987,30.196,155.734
C08593=1051.013,-117.607,433.295,169.985,30.196,155.734
C08594=1051.007,-117.857,433.304,169.983,30.196,155.734
C08595=1051.000,-118.107,433.314,169.981,30.195,155.734
C08596=1050.994,-118.356,433.323,169.979,30.195,155.735
C08597=1050.989,-118.606,433.332,169.977,30.194,155.735
C08598=1050.983,-118.855,433.342,169.975,30.194,155.735
C08599=1050.976,-119.105,433.352,169.973,30.193,155.735
C08600=1050.970,-119.355,433.361,169.971,30.193,155.735
C08601=1050.964,-119.605,433.371,169.968,30.192,155.735
C08602=1050.957,-119.855,433.379,169.966,30.192,155.735
C08603=1050.951,-120.105,433.389,169.964,30.192,155.735
C08604=1050.946,-120.354,433.398,169.962,30.191,155.735
C08605=1050.939,-120.604,433.407,169.959,30.191,155.735
C08606=1050.933,-120.853,433.417,169.957,30.190,155.735
C08607=1050.927,-121.103,433.426,169.955,30.191,155.735
C08608=1050.921,-121.354,433.435,169.953,30.190,155.735
C08609=1050.915,-121.603,433.445,169.951,30.190,155.736
C08610=1050.909,-121.852,433.453,169.949,30.189,155.736
C08611=1050.903,-122.102,433.463,169.947,30.189,155.736
C08612=1050.896,-122.352,433.473,169.945,30.189,155.736
C08613=1050.891,-122.602,433.481,169.943,30.188,155.736
C08614=1050.884,-122.852,433.491,169.940,30.188,155.736
C08615=1050.879,-123.101,433.500,169.938,30.188,155.736
C08616=1050.872,-123.351,433.509,169.936,30.187,155.736
C08617=1050.866,-123.601,433.518,169.934,30.187,155.736
C08618=1050.860,-123.851,433.528,169.932,30.187,155.736
C08619=1050.854,-124.101,433.537,169.929,30.186,155.736
C08620=1050.848,-124.350,433.546,169.927,30.186,155.736
C08621=1050.842,-124.600,433.555,169.925,30.186,155.737
C08622=1050.835,-124.850,433.564,169.923,30.186,155.737
C08623=1050.829,-125.099,433.574,169.920,30.185,155.737
C08624=1050.823,-125.350,433.583,169.919,30.185,155.737
C08625=1050.817,-125.599,433.591,169.917,30.184,155.737
C08626=1050.811,-125.848,433.601,169.915,30.185,155.737
C08627=1050.805,-126.099,433.610,169.912,30.184,155.737
C08628=1050.798,-126.348,433.619,169.910,30.184,155.737
C08629=1050.793,-126.597,433.628,169.908,30.183,155.737
C08630=1050.787,-126.848,433.637,169.906,30.184,155.737
C08631=1050.780,-127.097,433.646,169.903,30.183,155.738
C08632=1050.774,-127.347,433.655,169.901,30.183,155.738
C08633=1050.768,-127.597,433.664,169.899,30.183,155.738
C08634=1050.762,-127.847,433.673,169.897,30.182,155.738
C08635=1050.758,-128.097,433.682,169.895,30.182,155.738
C08636=1050.754,-128.346,433.693,169.893,30.181,155.738
C08637=1050.750,-128.596,433.704,169.892,30.179,155.738
C08638=1050.748,-128.846,433.715,169.890,30.176,155.737
C08639=1050.747,-129.097,433.728,169.888,30.174,155.737
C08640=1050.747,-129.348,433.741,169.886,30.171,155.737
C08641=1050.749,-129.598,433.754,169.886,30.168,155.736
C08642=1050.751,-129.847,433.768,169.884,30.163,155.735
C08643=1050.754,-130.099,433.783,169.883,30.158,155.735
C08644=1050.760,-130.350,433.799,169.883,30.154,155.734
C08645=1050.764,-130.600,433.815,169.881,30.148,155.733
C08646=1050.771,-130.850,433.831,169.881,30.141,155.732
C08647=1050.406,-130.873,433.607,169.835,30.310,155.764
C08648=1050.400,-130.623,433.591,169.836,30.316,155.765
C08649=1050.395,-130.373,433.574,169.836,30.321,155.766
C08650=1050.389,-130.122,433.559,169.838,30.327,155.767
C08651=1050.386,-129.871,433.544,169.838,30.331,155.767
C08652=1050.384,-129.621,433.529,169.839,30.335,155.768
C08653=1050.382,-129.371,433.516,169.841,30.339,155.769
C08654=1050.382,-129.120,433.503,169.842,30.342,155.769
C08655=1050.383,-128.870,433.491,169.843,30.345,155.769
C08656=1050.385,-128.620,433.479,169.845,30.347,155.770
C08657=1050.388,-128.370,433.469,169.847,30.349,155.770
C08658=1050.391,-128.120,433.458,169.849,30.350,155.770
C08659=1050.396,-127.870,433.448,169.851,30.350,155.770
C08660=1050.403,-127.621,433.439,169.854,30.351,155.770
C08661=1050.409,-127.370,433.431,169.856,30.351,155.770
C08662=1050.415,-127.121,433.421,169.857,30.352,155.770
C08663=1050.421,-126.872,433.412,169.859,30.352,155.770
C08664=1050.427,-126.621,433.404,169.862,30.352,155.769
C08665=1050.433,-126.372,433.394,169.864,30.352,155.769
C08666=1050.439,-126.121,433.385,169.866,30.353,155.769
C08667=1050.445,-125.872,433.377,169.868,30.353,155.769
C08668=1050.451,-125.623,433.367,169.871,30.353,155.769
C08669=1050.457,-125.372,433.358,169.873,30.353,155.769
C08670=1050.464,-125.123,433.349,169.875,30.353,155.769
C08671=1050.470,-124.874,433.340,169.877,30.354,155.769
C08672=1050.476,-124.623,433.331,169.880,30.354,155.769
C08673=1050.482,-124.373,433.322,169.882,30.354,155.768
C08674=1050.489,-124.124,433.313,169.884,30.354,155.768
C08675=1050.495,-123.874,433.303,169.886,30.355,155.768
C08676=1050.500,-123.624,433.295,169.889,30.355,155.768
C08677=1050.506,-123.375,433.285,169.890,30.355,155.768
C08678=1050.513,-123.125,433.275,169.892,30.356,155.768
C08679=1050.519,-122.875,433.266,169.894,30.356,155.768
C08680=1050.525,-122.625,433.258,169.896,30.356,155.768
C08681=1050.531,-122.376,433.248,169.899,30.357,155.768
C08682=1050.537,-122.126,433.239,169.901,30.357,155.768
C08683=1050.543,-121.876,433.229,169.903,30.357,155.768
C08684=1050.549,-121.626,433.220,169.905,30.357,155.768
C08685=1050.555,-121.376,433.211,169.908,30.358,155.767
C08686=1050.562,-121.127,433.202,169.910,30.358,155.767
C08687=1050.568,-120.877,433.193,169.912,30.359,155.767
C08688=1050.574,-120.628,433.183,169.914,30.359,155.767
C08689=1050.580,-120.378,433.174,169.917,30.359,155.767
C08690=1050.586,-120.127,433.165,169.919,30.360,155.767
C08691=1050.592,-119.878,433.155,169.921,30.360,155.767
C08692=1050.598,-119.628,433.146,169.922,30.360,155.767
C08693=1050.604,-119.379,433.136,169.924,30.361,155.767
C08694=1050.611,-119.129,433.127,169.927,30.361,155.767
C08695=1050.617,-118.879,433.118,169.929,30.362,155.767
C08696=1050.623,-118.630,433.108,169.931,30.362,155.767
C08697=1050.629,-118.380,433.099,169.933,30.362,155.767
C08698=1050.635,-118.129,433.090,169.936,30.363,155.766
C08699=1050.641,-117.880,433.080,169.938,30.363,155.766
C08700=1050.647,-117.630,433.071,169.940,30.363,155.766
C08701=1050.653,-117.381,433.061,169.942,30.364,155.766
C08702=1050.659,-117.131,433.052,169.945,30.365,155.766
C08703=1050.665,-116.881,433.042,169.947,30.365,155.766
C08704=1050.672,-116.631,433.033,169.949,30.366,155.766
C08705=1050.678,-116.382,433.023,169.951,30.366,155.766
C08706=1050.684,-116.132,433.014,169.952,30.366,155.766
C08707=1050.690,-115.882,433.004,169.955,30.367,155.766
C08708=1050.697,-115.597,432.993,169.957,30.367,155.766
C08709=1050.704,-115.312,432.983,169.960,30.368,155.766
C08710=1050.712,-115.027,432.972,169.962,30.368,155.766
C08711=1050.718,-114.742,432.961,169.965,30.369,155.766
C08712=1050.724,-114.492,432.951,169.967,30.369,155.766
C08713=1050.730,-114.242,432.942,169.969,30.370,155.765
C08714=1050.737,-113.993,432.932,169.971,30.370,155.765
C08715=1050.743,-113.743,432.922,169.974,30.371,155.765
C08716=1050.749,-113.493,432.912,169.976,30.371,155.765
C08717=1050.755,-113.244,432.903,169.978,30.372,155.765
C08718=1050.761,-112.994,432.893,169.979,30.372,155.765
C08719=1050.768,-112.744,432.884,169.982,30.373,155.765
C08720=1050.774,-112.494,432.874,169.984,30.373,155.765
C08721=1050.779,-112.245,432.865,169.986,30.374,155.765
C08722=1050.786,-111.995,432.855,169.988,30.374,155.765
C08723=1050.792,-111.746,432.846,169.990,30.375,155.765
C08724=1050.798,-111.496,432.836,169.993,30.375,155.765
C08725=1050.804,-111.246,432.825,169.995,30.376,155.765
C08726=1050.810,-110.997,432.816,169.997,30.376,155.765
C08727=1050.816,-110.747,432.806,169.999,30.377,155.765
C08728=1050.822,-110.497,432.797,170.001,30.377,155.765
C08729=1050.828,-110.247,432.787,170.004,30.378,155.765
C08730=1050.834,-109.997,432.778,170.005,30.379,155.765
C08731=1050.841,-109.748,432.767,170.007,30.379,155.765
C08732=1050.847,-109.498,432.758,170.009,30.380,155.765
C08733=1050.853,-109.249,432.748,170.012,30.380,155.765
C08734=1050.859,-108.998,432.738,170.014,30.381,155.764
C08735=1050.866,-108.748,432.728,170.016,30.381,155.764
C08736=1050.872,-108.499,432.718,170.018,30.382,155.764
C08737=1050.878,-108.249,432.708,170.020,30.382,155.764
C08738=1050.884,-107.999,432.699,170.023,30.383,155.764
C08739=1050.891,-107.749,432.689,170.025,30.384,155.764
C08740=1050.897,-107.500,432.679,170.027,30.384,155.764
C08741=1050.903,-107.250,432.669,170.029,30.384,155.764
C08742=1050.909,-107.000,432.659,170.030,30.385,155.764
C08743=1050.915,-106.750,432.649,170.033,30.386,155.764
C08744=1050.921,-106.501,432.639,170.035,30.387,155.764
C08745=1050.927,-106.252,432.630,170.037,30.387,155.764
C08746=1050.933,-106.001,432.619,170.039,30.388,155.764
C08747=1050.939,-105.752,432.609,170.041,30.388,155.764
C08748=1050.946,-105.502,432.600,170.044,30.389,155.764
C08749=1050.952,-105.253,432.590,170.046,30.390,155.764
C08750=1050.957,-105.003,432.579,170.048,30.390,155.764
C08751=1050.964,-104.753,432.570,170.050,30.391,155.764
C08752=1050.970,-104.503,432.560,170.052,30.392,155.764
C08753=1050.976,-104.253,432.549,170.054,30.393,155.764
C08754=1050.982,-104.004,432.539,170.056,30.393,155.764
C08755=1050.989,-103.754,432.529,170.058,30.394,155.764
C08756=1050.995,-103.505,432.519,170.060,30.394,155.764
C08757=1051.000,-103.254,432.509,170.062,30.395,155.764
C08758=1051.007,-103.005,432.499,170.065,30.396,155.764
C08759=1051.013,-102.755,432.489,170.067,30.397,155.764
C08760=1051.019,-102.506,432.479,170.069,30.397,155.764
C08761=1051.026,-102.255,432.469,170.071,30.398,155.764
C08762=1051.032,-102.006,432.458,170.073,30.399,155.764
C08763=1051.037,-101.756,432.448,170.075,30.399,155.764
C08764=1051.044,-101.506,432.439,170.077,30.400,155.764
C08765=1051.050,-101.257,432.428,170.079,30.401,155.764
C08766=1051.056,-101.007,432.418,170.081,30.402,155.764
C08767=1051.062,-100.758,432.408,170.083,30.402,155.764
C08768=1051.069,-100.507,432.398,170.086,30.403,155.764
C08769=1051.074,-100.258,432.387,170.088,30.404,155.764
C08770=1051.081,-100.008,432.377,170.090,30.404,155.764
C08771=1051.087,-99.759,432.367,170.092,30.405,155.764
C08772=1051.093,-99.473,432.355,170.095,30.406,155.764
C08773=1051.101,-99.186,432.343,170.097,30.407,155.764
C08774=1051.108,-98.900,432.331,170.099,30.408,155.764
C08775=1051.115,-98.614,432.320,170.101,30.408,155.764
C08776=1051.121,-98.364,432.310,170.103,30.409,155.764
C08777=1051.128,-98.114,432.299,170.106,30.410,155.764
C08778=1051.134,-97.865,432.289,170.108,30.411,155.764
C08779=1051.140,-97.615,432.279,170.110,30.412,155.764
C08780=1051.146,-97.366,432.268,170.112,30.413,155.764
C08781=1051.152,-97.116,432.259,170.114,30.413,155.764
C08782=1051.158,-96.866,432.248,170.116,30.414,155.764
C08783=1051.164,-96.616,432.237,170.118,30.415,155.764
C08784=1051.170,-96.366,432.227,170.120,30.416,155.764
C08785=1051.176,-96.117,432.216,170.122,30.417,155.764
C08786=1051.183,-95.868,432.206,170.124,30.417,155.764
C08787=1051.189,-95.617,432.195,170.126,30.418,155.764
C08788=1051.195,-95.368,432.185,170.128,30.419,155.764
C08789=1051.201,-95.118,432.174,170.131,30.420,155.764
C08790=1051.206,-94.868,432.164,170.133,30.421,155.764
C08791=1051.213,-94.619,432.154,170.135,30.422,155.764
C08792=1051.219,-94.369,432.143,170.137,30.422,155.764
C08793=1051.225,-94.119,432.133,170.138,30.423,155.764
C08794=1051.231,-93.869,432.122,170.140,30.424,155.764
C08795=1051.237,-93.620,432.111,170.143,30.425,155.764
C08796=1051.244,-93.370,432.101,170.145,30.426,155.764
C08797=1051.249,-93.120,432.090,170.147,30.427,155.764
C08798=1051.256,-92.871,432.080,170.149,30.428,155.764
C08799=1051.261,-92.621,432.069,170.151,30.429,155.764
C08800=1051.268,-92.371,432.058,170.153,30.430,155.764
C08801=1051.274,-92.122,432.048,170.156,30.431,155.764
C08802=1051.280,-91.872,432.038,170.157,30.432,155.764
C08803=1051.285,-91.622,432.027,170.159,30.433,155.764
C08804=1051.293,-91.372,432.016,170.161,30.434,155.764
C08805=1051.298,-91.123,432.005,170.163,30.434,155.764
C08806=1051.304,-90.873,431.994,170.165,30.435,155.764
C08807=1051.311,-90.623,431.984,170.168,30.436,155.764
C08808=1051.317,-90.373,431.973,170.170,30.437,155.764
C08809=1051.323,-90.124,431.963,170.172,30.438,155.764
C08810=1051.329,-89.874,431.952,170.174,30.439,155.764
C08811=1051.335,-89.625,431.941,170.175,30.440,155.764
C08812=1051.342,-89.375,431.931,170.177,30.441,155.764
C08813=1051.348,-89.125,431.920,170.180,30.442,155.764
C08814=1051.353,-88.875,431.909,170.182,30.443,155.764
C08815=1051.360,-88.626,431.899,170.184,30.444,155.764
C08816=1051.366,-88.376,431.888,170.186,30.445,155.764
C08817=1051.372,-88.126,431.877,170.188,30.445,155.764
C08818=1051.378,-87.877,431.867,170.190,30.446,155.764
C08819=1051.385,-87.627,431.855,170.193,30.447,155.764
C08820=1051.390,-87.377,431.845,170.194,30.448,155.764
C08821=1051.397,-87.128,431.834,170.196,30.449,155.765
C08822=1051.403,-86.878,431.823,170.198,30.450,155.765
C08823=1051.409,-86.629,431.812,170.200,30.451,155.765
C08824=1051.416,-86.379,431.802,170.202,30.452,155.765
C08825=1051.422,-86.129,431.791,170.204,30.453,155.765
C08826=1051.428,-85.880,431.780,170.207,30.454,155.765
C08827=1051.435,-85.630,431.769,170.209,30.455,155.765
C08828=1051.440,-85.380,431.758,170.211,30.456,155.765
C08829=1051.447,-85.130,431.747,170.212,30.457,155.765
C08830=1051.453,-84.881,431.737,170.214,30.458,155.765
C08831=1051.459,-84.631,431.726,170.216,30.459,155.765
C08832=1051.465,-84.381,431.715,170.219,30.460,155.765
C08833=1051.471,-84.132,431.704,170.221,30.461,155.765
C08834=1051.478,-83.882,431.693,170.223,30.462,155.765
C08835=1051.484,-83.632,431.682,170.225,30.463,155.765
C08836=1051.491,-83.348,431.670,170.227,30.464,155.765
C08837=1051.498,-83.064,431.657,170.230,30.465,155.765
C08838=1051.506,-82.781,431.645,170.231,30.466,155.765
C08839=1051.513,-82.497,431.632,170.234,30.467,155.765
C08840=1051.518,-82.247,431.621,170.236,30.468,155.765
C08841=1051.525,-81.997,431.610,170.238,30.469,155.765
C08842=1051.531,-81.748,431.600,170.240,30.470,155.765
C08843=1051.538,-81.498,431.589,170.242,30.471,155.766
C08844=1051.543,-81.248,431.578,170.244,30.472,155.766
C08845=1051.550,-80.998,431.566,170.247,30.473,155.766
C08846=1051.556,-80.749,431.556,170.249,30.474,155.766
C08847=1051.563,-80.499,431.544,170.250,30.475,155.766
C08848=1051.569,-80.250,431.533,170.252,30.477,155.766
C08849=1051.576,-80.000,431.523,170.254,30.478,155.766
C08850=1051.581,-79.750,431.512,170.256,30.479,155.766
C08851=1051.588,-79.500,431.501,170.258,30.480,155.766
C08852=1051.594,-79.251,431.489,170.261,30.481,155.766
C08853=1051.600,-79.001,431.478,170.263,30.482,155.766
C08854=1051.606,-78.752,431.467,170.265,30.483,155.766
C08855=1051.612,-78.501,431.456,170.266,30.484,155.766
C08856=1051.618,-78.252,431.444,170.268,30.485,155.766
C08857=1051.625,-78.002,431.433,170.270,30.486,155.766
C08858=1051.630,-77.753,431.422,170.272,30.488,155.766
C08859=1051.637,-77.503,431.411,170.274,30.489,155.767
C08860=1051.643,-77.254,431.399,170.277,30.490,155.767
C08861=1051.649,-77.004,431.388,170.279,30.491,155.767
C08862=1051.655,-76.754,431.377,170.281,30.492,155.767
C08863=1051.661,-76.504,431.365,170.282,30.493,155.767
C08864=1051.667,-76.255,431.354,170.284,30.494,155.767
C08865=1051.674,-76.005,431.343,170.286,30.496,155.767
C08866=1051.680,-75.755,431.332,170.288,30.497,155.767
C08867=1051.686,-75.506,431.320,170.290,30.497,155.767
C08868=1051.692,-75.256,431.309,170.293,30.499,155.767
C08869=1051.698,-75.007,431.297,170.295,30.500,155.767
C08870=1051.705,-74.756,431.286,170.297,30.501,155.767
C08871=1051.710,-74.507,431.275,170.298,30.502,155.767
C08872=1051.717,-74.257,431.263,170.300,30.504,155.767
C08873=1051.723,-74.007,431.252,170.302,30.505,155.768
C08874=1051.729,-73.758,431.241,170.304,30.506,155.768
C08875=1051.736,-73.508,431.229,170.306,30.507,155.768
C08876=1051.741,-73.259,431.218,170.308,30.508,155.768
C08877=1051.748,-73.009,431.206,170.311,30.510,155.768
C08878=1051.753,-72.759,431.195,170.313,30.511,155.768
C08879=1051.760,-72.510,431.183,170.314,30.512,155.768
C08880=1051.766,-72.260,431.172,170.316,30.513,155.768
C08881=1051.772,-72.011,431.160,170.318,30.515,155.768
C08882=1051.777,-71.761,431.148,170.320,30.516,155.768
C08883=1051.784,-71.511,431.136,170.322,30.517,155.769
C08884=1051.790,-71.261,431.125,170.324,30.518,155.769
C08885=1051.796,-71.012,431.114,170.326,30.520,155.769
C08886=1051.803,-70.762,431.102,170.328,30.521,155.769
C08887=1051.808,-70.513,431.090,170.329,30.522,155.769
C08888=1051.814,-70.263,431.079,170.332,30.524,155.769
C08889=1051.821,-70.013,431.067,170.334,30.525,155.769
C08890=1051.827,-69.764,431.056,170.336,30.526,155.769
C08891=1051.832,-69.514,431.044,170.338,30.527,155.769
C08892=1051.838,-69.264,431.033,170.340,30.529,155.769
C08893=1051.845,-69.015,431.021,170.342,30.530,155.770
C08894=1051.851,-68.765,431.008,170.343,30.531,155.770
C08895=1051.857,-68.515,430.997,170.345,30.532,155.770
C08896=1051.863,-68.266,430.985,170.347,30.534,155.770
C08897=1051.869,-68.016,430.974,170.349,30.535,155.770
C08898=1051.875,-67.766,430.962,170.351,30.536,155.770
C08899=1051.881,-67.517,430.950,170.353,30.538,155.770
C08900=1051.888,-67.235,430.937,170.356,30.539,155.770
C08901=1051.895,-66.953,430.924,170.358,30.541,155.770
C08902=1051.902,-66.672,430.911,170.360,30.542,155.771
C08903=1051.909,-66.390,430.897,170.362,30.544,155.771
C08904=1051.915,-66.139,430.886,170.364,30.545,155.771
C08905=1051.921,-65.891,430.874,170.366,30.546,155.771
C08906=1051.927,-65.641,430.862,170.368,30.547,155.771
C08907=1051.934,-65.391,430.850,170.370,30.549,155.771
C08908=1051.940,-65.142,430.839,170.372,30.551,155.771
C08909=1051.945,-64.892,430.826,170.373,30.551,155.771
C08910=1051.952,-64.642,430.814,170.375,30.553,155.771
C08911=1051.958,-64.392,430.803,170.378,30.554,155.771
C08912=1051.964,-64.143,430.791,170.380,30.556,155.772
C08913=1051.970,-63.893,430.779,170.382,30.557,155.772
C08914=1051.977,-63.644,430.767,170.384,30.558,155.772
C08915=1051.983,-63.394,430.756,170.386,30.560,155.772
C08916=1051.989,-63.144,430.744,170.388,30.561,155.772
C08917=1051.995,-62.895,430.732,170.389,30.562,155.772
C08918=1052.002,-62.645,430.720,170.391,30.564,155.772
C08919=1052.007,-62.395,430.708,170.393,30.565,155.773
C08920=1052.014,-62.146,430.696,170.395,30.566,155.773
C08921=1052.020,-61.896,430.684,170.397,30.568,155.773
C08922=1052.026,-61.646,430.672,170.399,30.569,155.773
C08923=1052.033,-61.397,430.660,170.401,30.570,155.773
C08924=1052.039,-61.147,430.649,170.402,30.572,155.773
C08925=1052.045,-60.897,430.636,170.405,30.573,155.773
C08926=1052.051,-60.648,430.624,170.407,30.575,155.773
C08927=1052.058,-60.398,430.612,170.409,30.576,155.773
C08928=1052.064,-60.148,430.600,170.411,30.577,155.773
C08929=1052.070,-59.900,430.588,170.413,30.579,155.774
C08930=1052.076,-59.650,430.576,170.415,30.580,155.774
C08931=1052.082,-59.399,430.564,170.417,30.582,155.774
C08932=1052.089,-59.150,430.553,170.418,30.583,155.774
C08933=1052.095,-58.900,430.540,170.420,30.584,155.774
C08934=1052.101,-58.651,430.528,170.422,30.586,155.774
C08935=1052.107,-58.402,430.516,170.424,30.587,155.774
C08936=1052.113,-58.152,430.504,170.426,30.588,155.775
C08937=1052.120,-57.902,430.492,170.428,30.590,155.775
C08938=1052.126,-57.653,430.480,170.430,30.591,155.775
C08939=1052.132,-57.403,430.467,170.431,30.592,155.775
C08940=1052.139,-57.153,430.455,170.433,30.594,155.775
C08941=1052.144,-56.904,430.443,170.436,30.596,155.775
C08942=1052.151,-56.654,430.431,170.438,30.597,155.775
C08943=1052.158,-56.405,430.419,170.440,30.598,155.775
C08944=1052.164,-56.155,430.407,170.442,30.600,155.776
C08945=1052.170,-55.905,430.395,170.444,30.601,155.776
C08946=1052.177,-55.656,430.383,170.446,30.602,155.776
C08947=1052.183,-55.406,430.370,170.447,30.604,155.776
C08948=1052.189,-55.156,430.358,170.449,30.605,155.776
C08949=1052.195,-54.906,430.346,170.451,30.606,155.776
C08950=1052.202,-54.657,430.334,170.453,30.608,155.776
C08951=1052.208,-54.408,430.322,170.455,30.609,155.776
C08952=1052.214,-54.158,430.310,170.457,30.611,155.777
C08953=1052.221,-53.908,430.298,170.459,30.612,155.777
C08954=1052.226,-53.659,430.285,170.460,30.613,155.777
C08955=1052.233,-53.409,430.273,170.462,30.615,155.777
C08956=1052.240,-53.159,430.261,170.464,30.616,155.777
C08957=1052.246,-52.910,430.249,170.466,30.617,155.777
C08958=1052.252,-52.660,430.237,170.468,30.619,155.777
C08959=1052.258,-52.410,430.224,170.470,30.620,155.778
C08960=1052.265,-52.161,430.212,170.472,30.622,155.778
C08961=1052.271,-51.911,430.200,170.474,30.624,155.778
C08962=1052.278,-51.662,430.187,170.476,30.625,155.778
C08963=1052.284,-51.412,430.175,170.478,30.626,155.778
C08964=1052.291,-51.131,430.161,170.480,30.628,155.778
C08965=1052.299,-50.851,430.148,170.482,30.629,155.778
C08966=1052.305,-50.570,430.133,170.484,30.631,155.779
C08967=1052.312,-50.290,430.119,170.487,30.633,155.779
C08968=1052.319,-50.040,430.107,170.488,30.634,155.779
C08969=1052.325,-49.791,430.094,170.490,30.636,155.779
C08970=1052.331,-49.541,430.082,170.492,30.637,155.779
C08971=1052.337,-49.291,430.069,170.494,30.639,155.779
C08972=1052.343,-49.042,430.057,170.496,30.640,155.779
C08973=1052.349,-48.793,430.044,170.498,30.642,155.780
C08974=1052.355,-48.543,430.032,170.500,30.643,155.780
C08975=1052.361,-48.293,430.019,170.501,30.645,155.780
C08976=1052.368,-48.044,430.007,170.503,30.646,155.780
C08977=1052.374,-47.794,429.994,170.505,30.648,155.780
C08978=1052.380,-47.544,429.981,170.507,30.650,155.780
C08979=1052.386,-47.295,429.969,170.509,30.651,155.781
C08980=1052.392,-47.046,429.956,170.511,30.653,155.781
C08981=1052.398,-46.796,429.944,170.513,30.655,155.781
C08982=1052.404,-46.546,429.931,170.514,30.656,155.781
C08983=1052.411,-46.297,429.918,170.516,30.658,155.781
C08984=1052.417,-46.047,429.906,170.518,30.659,155.781
C08985=1052.423,-45.797,429.893,170.520,30.661,155.782
C08986=1052.429,-45.548,429.880,170.522,30.663,155.782
C08987=1052.435,-45.298,429.867,170.524,30.664,155.782
C08988=1052.442,-45.048,429.855,170.526,30.666,155.782
C08989=1052.448,-44.799,429.842,170.527,30.667,155.782
C08990=1052.454,-44.549,429.830,170.529,30.669,155.782
C08991=1052.460,-44.300,429.816,170.531,30.670,155.783
C08992=1052.466,-44.050,429.804,170.533,30.672,155.783
C08993=1052.473,-43.800,429.792,170.535,30.673,155.783
C08994=1052.479,-43.551,429.779,170.537,30.675,155.783
C08995=1052.485,-43.301,429.766,170.539,30.676,155.783
C08996=1052.492,-43.051,429.752,170.540,30.678,155.783
C08997=1052.498,-42.801,429.740,170.542,30.680,155.784
C08998=1052.505,-42.553,429.727,170.544,30.682,155.784
C08999=1052.510,-42.303,429.715,170.546,30.683,155.784
C09000=1052.516,-42.053,429.702,170.548,30.685,155.784
C09001=1052.523,-41.804,429.689,170.550,30.686,155.784
C09002=1052.528,-41.554,429.676,170.552,30.688,155.785
C09003=1052.535,-41.305,429.663,170.553,30.689,155.785
C09004=1052.541,-41.055,429.651,170.555,30.691,155.785
C09005=1052.548,-40.806,429.638,170.557,30.693,155.785
C09006=1052.553,-40.556,429.625,170.559,30.694,155.785
C09007=1052.560,-40.306,429.611,170.561,30.696,155.785
C09008=1052.566,-40.056,429.599,170.563,30.698,155.786
C09009=1052.573,-39.807,429.586,170.565,30.699,155.786
C09010=1052.579,-39.558,429.573,170.566,30.701,155.786
C09011=1052.585,-39.308,429.560,170.568,30.702,155.786
C09012=1052.591,-39.058,429.547,170.570,30.704,155.786
C09013=1052.597,-38.809,429.535,170.572,30.705,155.786
C09014=1052.604,-38.559,429.521,170.574,30.707,155.787
C09015=1052.610,-38.309,429.508,170.576,30.709,155.787
C09016=1052.616,-38.059,429.495,170.578,30.711,155.787
C09017=1052.623,-37.810,429.482,170.579,30.712,155.787
C09018=1052.628,-37.560,429.469,170.581,30.714,155.787
C09019=1052.635,-37.311,429.456,170.583,30.716,155.788
C09020=1052.641,-37.062,429.443,170.584,30.717,155.788
C09021=1052.647,-36.812,429.430,170.586,30.719,155.788
C09022=1052.653,-36.563,429.417,170.588,30.720,155.788
C09023=1052.660,-36.313,429.403,170.590,30.723,155.788
C09024=1052.666,-36.063,429.391,170.591,30.724,155.789
C09025=1052.672,-35.814,429.377,170.593,30.726,155.789
C09026=1052.678,-35.564,429.364,170.595,30.728,155.789
C09027=1052.684,-35.314,429.352,170.597,30.729,155.789
C09028=1052.691,-35.034,429.337,170.599,30.731,155.789
C09029=1052.697,-34.754,429.322,170.602,30.733,155.790
C09030=1052.705,-34.474,429.307,170.603,30.735,155.790
C09031=1052.712,-34.194,429.292,170.605,30.737,155.790
C09032=1052.718,-33.944,429.279,170.607,30.738,155.790
C09033=1052.724,-33.695,429.265,170.609,30.741,155.790
C09034=1052.730,-33.446,429.252,170.611,30.742,155.791
C09035=1052.737,-33.195,429.239,170.613,30.744,155.791
C09036=1052.743,-32.946,429.226,170.615,30.746,155.791
C09037=1052.749,-32.697,429.213,170.616,30.747,155.791
C09038=1052.755,-32.448,429.199,170.618,30.749,155.791
C09039=1052.761,-32.198,429.187,170.620,30.751,155.792
C09040=1052.768,-31.948,429.173,170.622,30.753,155.792
C09041=1052.774,-31.698,429.159,170.624,30.754,155.792
C09042=1052.780,-31.449,429.146,170.625,30.756,155.792
C09043=1052.786,-31.200,429.133,170.627,30.758,155.792
C09044=1052.793,-30.950,429.119,170.628,30.759,155.793
C09045=1052.799,-30.700,429.107,170.630,30.761,155.793
C09046=1052.805,-30.450,429.093,170.632,30.763,155.793
C09047=1052.811,-30.201,429.080,170.634,30.764,155.793
C09048=1052.818,-29.951,429.066,170.636,30.767,155.794
C09049=1052.824,-29.702,429.053,170.638,30.768,155.794
C09050=1052.830,-29.452,429.039,170.640,30.770,155.794
C09051=1052.836,-29.203,429.026,170.641,30.772,155.794
C09052=1052.843,-28.953,429.012,170.643,30.773,155.794
C09053=1052.849,-28.703,429.000,170.645,30.775,155.794
C09054=1052.855,-28.454,428.987,170.647,30.777,155.795
C09055=1052.862,-28.204,428.973,170.649,30.779,155.795
C09056=1052.868,-27.955,428.960,170.651,30.780,155.795
C09057=1052.874,-27.706,428.946,170.652,30.782,155.795
C09058=1052.880,-27.455,428.932,170.653,30.784,155.796
C09059=1052.886,-27.206,428.919,170.655,30.785,155.796
C09060=1052.893,-26.957,428.906,170.657,30.787,155.796
C09061=1052.899,-26.707,428.892,170.659,30.789,155.796
C09062=1052.905,-26.457,428.878,170.661,30.791,155.796
C09063=1052.911,-26.208,428.865,170.663,30.792,155.797
C09064=1052.917,-25.959,428.852,170.664,30.795,155.797
C09065=1052.923,-25.708,428.837,170.666,30.796,155.797
C09066=1052.930,-25.459,428.824,170.668,30.798,155.797
C09067=1052.936,-25.210,428.811,170.670,30.800,155.797
C09068=1052.942,-24.960,428.797,170.672,30.802,155.798
C09069=1052.948,-24.710,428.783,170.674,30.804,155.798
C09070=1052.954,-24.461,428.770,170.676,30.806,155.798
C09071=1052.960,-24.212,428.756,170.676,30.807,155.798
C09072=1052.967,-23.962,428.743,170.678,30.809,155.799
C09073=1052.973,-23.713,428.729,170.680,30.811,155.799
C09074=1052.979,-23.463,428.715,170.682,30.813,155.799
C09075=1052.985,-23.213,428.701,170.684,30.814,155.799
C09076=1052.991,-22.964,428.687,170.686,30.817,155.800
C09077=1052.997,-22.715,428.674,170.688,30.818,155.800
C09078=1053.004,-22.465,428.660,170.689,30.820,155.800
C09079=1053.009,-22.215,428.646,170.691,30.822,155.800
C09080=1053.016,-21.965,428.633,170.693,30.824,155.800
C09081=1053.022,-21.716,428.618,170.694,30.825,155.801
C09082=1053.028,-21.467,428.605,170.696,30.827,155.801
C09083=1053.035,-21.217,428.591,170.698,30.829,155.801
C09084=1053.040,-20.967,428.577,170.699,30.831,155.801
C09085=1053.047,-20.718,428.564,170.701,30.833,155.802
C09086=1053.053,-20.468,428.550,170.703,30.835,155.802
C09087=1053.059,-20.219,428.536,170.705,30.837,155.802
C09088=1053.066,-19.969,428.522,170.707,30.838,155.802
C09089=1053.072,-19.720,428.509,170.709,30.841,155.803
C09090=1053.078,-19.470,428.495,170.711,30.842,155.803
C09091=1053.084,-19.221,428.480,170.711,30.844,155.803
C09092=1053.092,-18.940,428.465,170.714,30.846,155.803
C09093=1053.098,-18.659,428.450,170.716,30.848,155.803
C09094=1053.105,-18.378,428.434,170.718,30.850,155.804
C09095=1053.112,-18.097,428.418,170.720,30.852,155.804
C09096=1053.118,-17.848,428.405,170.722,30.854,155.804
C09097=1053.125,-17.599,428.391,170.723,30.856,155.804
C09098=1053.131,-17.349,428.377,170.725,30.858,155.805
C09099=1053.138,-17.099,428.363,170.727,30.860,155.805
C09100=1053.143,-16.850,428.349,170.728,30.862,155.805
C09101=1053.150,-16.600,428.335,170.730,30.864,155.805
C09102=1053.156,-16.351,428.321,170.732,30.865,155.806
